IF NOT doPublish THEN
	LastPublished := 0;
	FOR i := 0 TO UsedPublishFbs - 1 DO
		PublishSendBools[i] := FALSE;
		Publishs[i](
	send:= PublishSendBools[i]);
	PublishSendFree[i] := TRUE;
	END_FOR
	
END_IF

MQTT_IN_OUT.clientFB(
	MQTT_IN_OUT:= MQTT_IN_OUT, 
	ENABLE:= TRUE, 
	URL:= broker, 
	TIMEOUT:= T#5S, 
	TLS:= FALSE);
start(CLK := working);

IF start.Q THEN
	finished := FALSE;

END_IF
IF doPublish THEN

	FOR i := 0 TO UsedPublishFbs - 1 DO
		
		IF PublishSendFree[i] AND NOT finished THEN
			PublishSendFree[i] := FALSE;
			
			//get next element
			IF LastPublished >= CountArray THEN
				finished := TRUE;
	
			ELSE
				IF TopicFix THEN
					PublishTopicStore[i] := Topic;
				ELSE
					PublishTopicStore[i] := Topic[LastPublished];	
				END_IF
				
				IF PayloadFix THEN
					PublishPayloadStore[i] := Payload;
				ELSE
					PublishPayloadStore[i] := Payload[LastPublished];	
				END_IF
				
				PublishSendBools[i] := TRUE;
			END_IF
			LastPublished := LastPublished + 1;
			
		END_IF	
		
			Publishs[i](
		Topic:=PublishTopicStore[i], 
		PayloadString:= PublishPayloadStore[i], 
		PublishAsString:= TRUE, 
		QoSIn:= QoS, 
		MRetain:= RetainIn, 
		send:= PublishSendBools[i]);
		IF Publishs[i].done THEN 
			PublishSendFree[i] := TRUE;
		END_IF
		IF Publishs[i].sendActive THEN
			PublishSendBools[i] := FALSE;
		END_IF
	END_FOR
	
END_IF

END_FUNCTION_BLOCK

// MQTT/Function/InitMQTTValue
FUNCTION InitMQTTValue : bool
VAR_INPUT
DataArray:POINTER TO CommonTypesAndFunctions.PWConfigs;
CountOfArray:UINT;
ValueToMQTTArray:POINTER TO MQTTValue;
MQTT_IN_OUT: POINTER TO MQTT_IN_OUT;
END_VAR
VAR
	i:UINT;
END_VAR

FOR i := 0 TO CountOfArray - 1 DO
	IF DataArray[i].NeedsMQTT THEN
		ValueToMQTTArray[i].Init(
			Topic:= DataArray[i].MQTTTopic, 
			ValueName:= DataArray[i].MQTTName, 
			ValuePointer:= DataArray[i].PointerTo, 
			ValueType:= DataArray[i].ValueType, 
			ValueDiff:= DataArray[i].MQTTDiff, 
			DecimalPlace:= DataArray[i].MQTTDezimal, 
			QoS:= DataArray[i].MQTTQoS, 
			RetainMqtt:= DataArray[i].MQTTRetain, 
			MinTime:= DataArray[i].MQTTTime,
			MQTT_IN_OUT:= MQTT_IN_OUT);
	END_IF
END_FOR

END_FUNCTION

// MQTT/Function Blocks/MQTTPushover
FUNCTION_BLOCK MQTTPushover
VAR_INPUT
	Data:POINTER TO PUSHOVER_DATA;
	MQTT_IN_OUT:REFERENCE TO MQTT_IN_OUT;
	CountData:UINT;
	MQTTTopic:POINTER TO STRING;
END_VAR
VAR_OUTPUT
END_VAR
VAR
	i:UINT;
	HaveToPush:BOOL;
	 
	Publish:MqttPublish;
	init:BOOL;
	PushedElement:UINT;
	SendFree: BOOL;
	// at least one message to push
	hit: BOOL;
	hitIndex:UINT;
	(*build like 'Topic(n(x)):x, Payload(n(x):x, Prio:x, Sound:x'  *)
	SendString:STRING(500);
	tmpString:STRING;
END_VAR

IF NOT init THEN
	
	init := TRUE;
	Publish.SetMqttInOut(MQTT_IN_OUT:= MQTT_IN_OUT);
END_IF
hit := FALSE;
HaveToPush := FALSE;
FOR i := 0 TO CountData - 1 DO
	IF Data[i].IsConfig THEN
		Data[i].R_T(CLK:=Data[i].Trigger^ XOR Data[i].Negate);
		IF Data[i].R_T.Q THEN
			Data[i].NeedToPush := TRUE;
		END_IF
		IF Data[i].NeedToPush THEN
			HaveToPush := TRUE;
		END_IF
		IF HaveToPush and NOT hit THEN
			hit := TRUE;
			hitIndex := i;
		END_IF
	END_IF
END_FOR

IF Publish.done THEN
	SendFree := TRUE;
END_IF


IF HaveToPush AND SendFree THEN
	SendFree := FALSE;
	//now build message
	SendString := 'Topic(';
	//add topic length
	tmpString := TO_STRING(len(Data[hitIndex].Topic^));
 	CommonTypesAndFunctions.concat(s1:= ADR(SendString), S2:=ADR(tmpString));
	//add '):'
	CommonTypesAndFunctions.concat(s1:= ADR(SendString), S2:=ADR('):'));
	//add topic
	CommonTypesAndFunctions.concat(s1:= ADR(SendString), S2:=Data[hitIndex].Topic);
	//add fixtext
	CommonTypesAndFunctions.concat(s1:= ADR(SendString), S2:=ADR(', Payload('));
	//add payload length
	tmpString := TO_STRING(len(Data[hitIndex].Payload^));
 	CommonTypesAndFunctions.concat(s1:= ADR(SendString), S2:=ADR(tmpString));
	//add '):'
	CommonTypesAndFunctions.concat(s1:= ADR(SendString), S2:=ADR('):'));
	//add topic
	CommonTypesAndFunctions.concat(s1:= ADR(SendString), S2:=Data[hitIndex].Payload);
	//add fixtext
	CommonTypesAndFunctions.concat(s1:= ADR(SendString), S2:=ADR(', Prio:'));
	//add prio
	tmpString := TO_STRING(Data[hitIndex].Prio);
 	CommonTypesAndFunctions.concat(s1:= ADR(SendString), S2:=ADR(tmpString));
	//add fixtext
	CommonTypesAndFunctions.concat(s1:= ADR(SendString), S2:=ADR(', Sound:'));
	//add prio
	tmpString := TO_STRING(Data[hitIndex].Sound);
 	CommonTypesAndFunctions.concat(s1:= ADR(SendString), S2:=ADR(tmpString));
	//done
	Data[hitIndex].NeedToPush := FALSE;
	//now send
	
END_IF

Publish(
	Topic:= MQTTTopic, 
	PayloadString:= adr(SendString), 
	PublishAsString:= TRUE, 
	QoSIn:= QoS.ExactlyOnce, 
	MRetain:= true, 
	send:= NOT SendFree);

END_FUNCTION_BLOCK

// MQTT/Function Blocks/CallbackFBs/SingelCallbacks/SingelStringCallback
FUNCTION_BLOCK SingelStringCallback IMPLEMENTS MQTT_SUBSCRIBE_CALLBACK
VAR_INPUT
END_VAR
VAR_OUTPUT
	//data was received, you have to reset this bit after checking!
	received: BOOL;
END_VAR
VAR
	MyPayload : POINTER TO STRING;
	MyTopic : POINTER TO STRING;
END_VAR

METHOD PublishReceived : BOOL
VAR_INPUT
	//Collection of received Data
	Data:CALLBACK_DATA;

END_VAR
MEM.MemMove(pSource:= Data.PayloadString, pDestination:= MyPayload, uiNumberOfBytes:= TO_UINT(data.PayloadSize + 1));
MEM.MemMove(pSource:= Data.TopicOut, pDestination:= MyTopic, uiNumberOfBytes:= CommonTypesAndFunctions.len(Data.TopicOut) + 1);

received := TRUE;
END_METHOD

METHOD Init : BOOL
VAR_INPUT
	payload:POINTER TO STRING;
	topic:POINTER TO STRING;
END_VAR
MyTopic := topic;
MyPayload := payload;
END_METHOD

METHOD ResetReceived : BOOL
VAR_INPUT
END_VAR
received := FALSE;
END_METHOD

END_FUNCTION_BLOCK

// MQTT/Function Blocks/CallbackFBs/SingelCallbacks/AllValuesCallback
(*
this FB expects all values as a string, binary receive is not suported...
Payload content is only value, no description, no special characters...
*)
FUNCTION_BLOCK AllValuesCallback IMPLEMENTS MQTT_SUBSCRIBE_CALLBACK
VAR_INPUT
END_VAR
VAR_OUTPUT
	//data was received, you have to reset this bit after checking!
	received: BOOL;

END_VAR
VAR
	VarType:IBaseLibrary.TypeClass;
	MyTarget:CommonTypesAndFunctions.ALL_TYPES_UNION_POINTER;
END_VAR

METHOD PublishReceived : BOOL
VAR_INPUT
	//Collection of received Data
	Data:CALLBACK_DATA;

END_VAR
CommonTypesAndFunctions.GetValueFromStringPt(TypeOfValue:= VarType,Target:= MyTarget, str:= DATA.PayloadString);

received := TRUE;
END_METHOD

METHOD Init : BOOL
VAR_INPUT
	SetType:IBaseLibrary.TypeClass;
	Target:CommonTypesAndFunctions.ALL_TYPES_UNION_POINTER;
END_VAR
VarType := SetType;
MyTarget := Target;
END_METHOD

METHOD ResetReceived : BOOL
VAR_INPUT
END_VAR
received := FALSE;
END_METHOD

END_FUNCTION_BLOCK

// MQTT/Function Blocks/CallbackFBs/ListCallbacks/ListAllValuesCallback
(*
this FB expects all values as a string, binary receive is not suported...
Payload content is only value, no description, no special characters...
*)
FUNCTION_BLOCK ListAllValuesCallback IMPLEMENTS MQTT_SUBSCRIBE_CALLBACK
VAR_INPUT
END_VAR
VAR_OUTPUT
END_VAR
VAR
	MyListData:POINTER TO LIST_ALLVALUES_CALLBACK_DATA;
	MyLengthOfData:ULINT;
	ListSplitTopic:BOOL;
	ListSplitPayload:BOOL;
	SplitCharPayload:BYTE;
END_VAR

METHOD PublishReceived : BOOL
VAR_INPUT
	//Collection of received Data
	Data:CALLBACK_DATA;
END_VAR

VAR
	i:ULINT;
	StrPt:POINTER TO STRING;
END_VAR
IF ListSplitTopic THEN
	//now search the right topic 
	FOR i := 0 TO MyLengthOfData - 1 DO
		IF CommonTypesAndFunctions.StrEquals(str1:= Data.TopicOutSplit^.Topics[Data.TopicOutSplit^.ValidFields - 1], str2:= MyListData[i].SubTopic) THEN
			CommonTypesAndFunctions.GetValueFromStringPt(TypeOfValue:= MyListData[i].VarTYPE ,Target:= MyListData[i].Target, str:= DATA.PayloadString);
		END_IF
	END_FOR
END_IF
IF ListSplitPayload THEN
	FOR i := 0 TO MyLengthOfData - 1 DO
		IF CommonTypesAndFunctions.StrEqualsAtStartWithDelimiter(str1:= MyListData[i].SubTopic, str2:= Data.PayloadString, delimiter:= SplitCharPayload) THEN
			//now search split char
			StrPt := Data.PayloadString;
			StrPt := StrPt + TO_DWORD(CommonTypesAndFunctions.find(str1 := StrPt, str2:= ADR(SplitCharPayload))) + 1;
			
			CommonTypesAndFunctions.GetValueFromStringPt(TypeOfValue:= MyListData[i].VarTYPE ,Target:= MyListData[i].Target, str:= StrPt);
		END_IF
	END_FOR
	
END_IF
END_METHOD

METHOD InitAsSplitTopic : BOOL
VAR_INPUT
	Data:POINTER TO LIST_ALLVALUES_CALLBACK_DATA;
	//Count of List Data
	LengthOfData:ULINT;
END_VAR
MyListData := Data;
MyLengthOfData := LengthOfData;
ListSplitTopic := TRUE;
ListSplitPayload := FALSE;
END_METHOD

(*inits FB, callback methoth then checks if the payload ist the same in the first characters as in the template
make sure to receive a string payload!
*)
METHOD InitAsSplitPayload : BOOL
VAR_INPUT
	Data:POINTER TO LIST_ALLVALUES_CALLBACK_DATA;
	//Count of List Data
	LengthOfData:ULINT;
	//spliting character
	SplitChar:BYTE;
END_VAR
MyListData :=Data;
MyLengthOfData := LengthOfData;
ListSplitTopic := FALSE;
ListSplitPayload := TRUE;
SplitCharPayload := SplitChar;
END_METHOD

END_FUNCTION_BLOCK

// MQTT/TestCases/testHighReceiveSplitPayload
FUNCTION_BLOCK testHighReceiveSplitPayload
VAR_INPUT
	Count:UINT:=TEST_TOPICS;
	broker:STRING:='test.mosquitto.org:1883';
	addTopic:STRING(200);
	repeatTime:TIME:=T#1M;
END_VAR
VAR_OUTPUT
END_VAR
VAR
	//MQTT_RECEIVE:MqttClient;
	
	
	subs:MQTTSubscribe;
	MQTT_IN_OUT_RECEIVE:MQTT_IN_OUT;
	tNewRun:TON;
	init: BOOL;
	i:UINT;
	//testTopics:ARRAY[0..TOPICS_MAX] OF STRING(255);
	testTopic:STRING:='SD_MQTT/TEST_PAYLOAD/PAYLOAD';
	testPayloadString:ARRAY[0..TOPICS_MAX]OF STRING(255);
	splitChar:STRING := '=';
	PayloadPrefix:STRING := 'Output';
	comparePayload:ARRAY[0..TOPICS_MAX]OF STRING(255);
	
	SendPayloadStorePointerArray:ARRAY[0..TOPICS_MAX] OF POINTER TO STRING;
	ReceivePayloadStore:ARRAY[0..TOPICS_MAX] OF LINT;
	SendPayloadStore:ARRAY[0..TOPICS_MAX] OF LINT;
	
	tmpString:STRING;
	tmpString2:STRING;
	step:UINT;
	subscribe: BOOL;

	HighSendPublish:HighLoadPublish;
	
	runPublishWorker: BOOL;

	
	noData: BOOL;
	nextRun: BOOL;
	ListCallback:ListAllValuesCallback;
	CallbackData:ARRAY[0..TOPICS_MAX] OF LIST_ALLVALUES_CALLBACK_DATA;
END_VAR
VAR CONSTANT
	TEST_TOPICS:UINT:= 200;
	TOPICS_MAX:UINT:=10000;
END_VAR

IF NOT init THEN
	init := TRUE;
	MQTT_IN_OUT_RECEIVE.ClientID := 'Test Client Receive';
	subs.SetMqttInOut(MQTT_IN_OUT:= MQTT_IN_OUT_RECEIVE); 
	//Testtopic();
	FOR i := 0 TO Count - 1 DO

		tmpString := PayloadPrefix;
		tmpString2 := UINT_TO_STRING(i);
		CommonTypesAndFunctions.concat(s1:= ADR(tmpString), s2:= ADR(tmpString2));
		//finished building compare payload
		comparePayload[i] := tmpString;
		CommonTypesAndFunctions.concat(s1:= ADR(tmpString), s2:= ADR(splitChar));
		SendPayloadStore[i] := i + 22;
		tmpString2 := TO_STRING(SendPayloadStore[i]);
		CommonTypesAndFunctions.concat(s1:= ADR(tmpString), s2:= ADR(tmpString2));
		//CommonTypesAndFunctions.concat(s1:= ADR(tmpString), s2:= ADR(splitChar));
		
		testPayloadString[i] := tmpString; 
		
		//compareTopic[i] := tmpString;
		CallbackData[i].SubTopic := ADR(comparePayload[i]);
		CallbackData[i].Target.POINTER_TO_LINT_T := ADR(ReceivePayloadStore[i]);
		CallbackData[i].VarTYPE := IBaseLibrary.TypeClass.TYPE_LINT;
		SendPayloadStorePointerArray[i] := ADR(testPayloadString[i]);
	END_FOR
	ListCallback.InitAsSplitPayload(Data:= ADR(CallbackData[0]), LengthOfData:= i, SplitChar:= CommonTypesAndFunctions.GetChar(splitChar));
END_IF
IF Count >= TOPICS_MAX THEN
	Count := TOPICS_MAX;
END_IF

subs(
	Subscribe:= subscribe, 
	Topic:= ADR(testTopic), 
	QoSSubscribe:= QoS.ExactlyOnce, 
	ExpectingString:= TRUE,
	Callback := ListCallback);
	
MQTT_IN_OUT_RECEIVE.clientFB(
	MQTT_IN_OUT:= MQTT_IN_OUT_RECEIVE, 
	ENABLE:= TRUE, 
	URL:= broker, 
	TIMEOUT:= T#5S, 
	TLS:= FALSE);
IF NOT MQTT_IN_OUT_RECEIVE.BROKER_CONNECTED THEN
	step := 0;
END_IF
	
HighSendPublish(
	ClientID:= 'HighSendClient', 
	Topic:= ADR(testTopic), 
	TopicFix:= TRUE, 
	payload:= ADR(SendPayloadStorePointerArray), 
	CountArray:= Count, 
	UsedPublishFbs:= 49, 
	working:= runPublishWorker, 
	broker:= broker, 
	QoS:= QoS.ExactlyOnce, 
	RetainIn:= FALSE);


CASE step OF
	0: 	step := 1;
		FOR i := 0 TO Count - 1 DO
			ReceivePayloadStore[i] := 0;
		END_FOR
	1: IF MQTT_IN_OUT_RECEIVE.BROKER_CONNECTED THEN
			step:= 5;
			//subscribe
			subscribe := TRUE;
		END_IF
	5: //wait for subscribe
		IF subs.SubscribeDone THEN
			step:= 10;
		END_IF
		 
	10: //publish all and receive data
		//start publish
		runPublishWorker := TRUE;
		step := 20;
	20: IF HighSendPublish.finished THEN
		//wait until send is done		
			runPublishWorker := FALSE;
			step:= 30;

		END_IF
	30: //now check payload
		
			noData := FALSE;
		FOR i := 0 TO Count - 1 DO
			IF ReceivePayloadStore[i] <> SendPayloadStore[i] THEN
				noData := TRUE;
				EXIT;
			END_IF
		END_FOR
		IF NOT noData THEN
			step := 40;
			//unsubscripe
			subscribe := FALSE; 
		END_IF	
	40: 
		IF nextRun OR tNewRun.Q THEN 
			nextRun := FALSE;
			step := 0;
		END_IF
END_CASE

tNewRun(in := step = 40,PT:= repeatTime);

END_FUNCTION_BLOCK

// MQTT/TestCases/testHighLoadPublish
FUNCTION_BLOCK testHighLoadPublish
VAR_INPUT
	topics:UINT:=TEST_TOPICS;
	broker:STRING:='test.mosquitto.org:1883';
	addTopic:STRING(200);
	retpeatTime:TIME:=T#1M;
END_VAR
VAR_OUTPUT
END_VAR
VAR

	HighLoad:HighLoadPublish;

	init: BOOL;
	i:UINT;
	//testTopics:ARRAY[0..TOPICS_MAX] OF STRING(255);
	testTopic:STRING(255):='High Payload Test with very very very very very very very very very very big topic/Outs';
	
	testPayload:ARRAY[0..TOPICS_MAX]OF STRING(255);
	splitChar:STRING := '=';
	PayloadPrefix:STRING := 'Output:';
	
	
	ReceivePayloadStore:ARRAY[0..TOPICS_MAX] OF LINT;
	SendPayloadStore:ARRAY[0..TOPICS_MAX] OF STRING(255);
	SendPayloadStorePointerArray:ARRAY[0..TOPICS_MAX] OF POINTER TO STRING;
	tmpString:STRING;
	tmpString2:STRING;
	step:INT;
	nextRun: BOOL;
	tNewRun:ton;
	work:BOOL;


END_VAR
VAR CONSTANT
	TEST_TOPICS:UINT:= 200;
	TOPICS_MAX:UINT:=10000;
END_VAR

IF NOT init THEN
	 init := TRUE;
	//Testtopic();
	FOR i := 0 TO topics - 1 DO
		
		tmpString := PayloadPrefix;
		tmpString2 := UINT_TO_STRING(i);
		CommonTypesAndFunctions.concat(s1:= ADR(tmpString), s2:= ADR(tmpString2));
		
		CommonTypesAndFunctions.concat(s1:= ADR(tmpString), s2:= ADR(splitChar));
		CommonTypesAndFunctions.concat(s1:= ADR(tmpString), s2:= ADR(tmpString2));
		SendPayloadStore[i] := tmpString;
		SendPayloadStorePointerArray[i] := ADR(SendPayloadStore[i]);
		step := 10;
	END_FOR
	
END_IF

HighLoad(
	ClientID:= 'Test for HighLoadPublish', 
	Topic:= ADR(testTopic), 
	TopicFix:= TRUE, 
	payload:= ADR(SendPayloadStorePointerArray[0]),
	PayloadFix := FALSE, 
	CountArray:= topics, 
	UsedPublishFbs:= MyConstants.IN_OUT_SLOTS_SIZE - 1, 
	working:= work, 
	broker:= 'windows-10-pro:1883', 
	QoS:= QoS.ExactlyOnce, 
	RetainIn:= FALSE);

IF topics >= TOPICS_MAX THEN
	topics := TOPICS_MAX - 1;
END_IF


	
CASE step OF
	10: //empty
		step := 20;
	
	20: 
		work := TRUE; 
		step := 30;
	30: //wait for finish
		IF HighLoad.finished THEN
			work := FALSE;
			step := 40;
			
		END_IF
		
	40: //wait for next run
		IF tNewRun.Q OR nextRun THEN
			step := 10;
		END_IF 
END_CASE

tNewRun(in := step = 40,PT:= retpeatTime);

END_FUNCTION_BLOCK

// MQTT/Function Blocks/CallbackFBs/Callback Collector/CallbackCollector
(*this FB collects instances of FB with the MQTT_SUBSCRIBE_CALLBACK interface.
then you can pass a instance of this FB to a subscription FB to call all of your FBs to a specific subscription topic,
in this call you can check if the packet was for your instance. If your instance methode call return true, the the FB exits the
loop an so you may save cycle time.
MEmory for instance references are created dynamic, so no restriction by library*)
FUNCTION_BLOCK CallbackCollector IMPLEMENTS MQTT_SUBSCRIBE_CALLBACK
VAR_INPUT
END_VAR
VAR_OUTPUT
END_VAR
VAR
	first:POINTER TO CALLBACK_INSTANCES := 0;
	items:UDINT;
	size:UDINT;
END_VAR

//true if all ok, else false
METHOD put : BOOL
VAR_INPUT
	instance:MQTT_SUBSCRIBE_CALLBACK;
END_VAR
VAR
	aktElement:POINTER TO CALLBACK_INSTANCES;
END_VAR
aktElement := first;

IF aktElement = 0 THEN
	//first hit...
	{info 'semaphore'}
	first := __NEW(CALLBACK_INSTANCES);
	IF first = 0 THEN
		put := FALSE;
		RETURN;
	END_IF
	aktElement := first;
ELSE
	//search last
	WHILE aktElement^.next  <> 0 DO 
		aktElement := aktElement^.next; 
	END_WHILE
	{info 'semaphore'}
	aktElement^.next := __NEW(CALLBACK_INSTANCES);
	IF aktElement^.next = 0 THEN
		put := FALSE;
		RETURN;
	END_IF
	aktElement := aktElement^.next;
END_IF

aktElement^.callback := instance;
put := TRUE;
items := items + 1;
size := size + SIZEOF(CALLBACK_INSTANCES);
END_METHOD


METHOD PublishReceived : BOOL
VAR_INPUT
	(*Collection of received Data*)
	Data	: CALLBACK_DATA;
END_VAR
VAR
	element:POINTER TO CALLBACK_INSTANCES;
	loop: BOOL := true;

END_VAR


IF first = 0 THEN
	//no callback avalable
	RETURN;
END_IF
element := first;


WHILE loop DO
	IF element^.callback.PublishReceived(Data := Data) THEN
		PublishReceived := TRUE;
		RETURN;
	END_IF
	IF element^.next = 0 THEN
		loop := FALSE;
	ELSE
		element := element^.next;
	END_IF
END_WHILE
END_METHOD

//destroy all dynamic content
METHOD destroy : BOOL
VAR_INPUT
END_VAR
VAR
	aktElement:POINTER TO CALLBACK_INSTANCES;
	nextElement:POINTER TO CALLBACK_INSTANCES;
	


END_VAR
GVL_MQTT.ProgNum := PROG_NUM.DESTROY_CALLBACK_COLLECTOR;
IF first = 0 THEN
	RETURN;
END_IF

aktElement := first;

REPEAT
	nextElement := aktElement^.next;
	__DELETE(aktElement);
	aktElement := nextElement;
	items := items - 1;
	size := size - SIZEOF(CALLBACK_INSTANCES);
UNTIL aktElement = 0
END_REPEAT
first := 0;
GVL_MQTT.ProgNum := PROG_NUM.DESTROY_CALLBACK_COLLECTOR_DONE;
END_METHOD

METHOD FB_Exit : BOOL 
VAR_INPUT 
 bInCopyCode : BOOL; // TRUE: the exit method is called in order to leave the instance which will be copied afterwards (online change). 
END_VAR
destroy();
END_METHOD

END_FUNCTION_BLOCK

// MQTT/TestCases/Test Interfaces/FooBarReceivingFB
{attribute 'reflection'}
FUNCTION_BLOCK FooBarReceivingFB IMPLEMENTS MQTT_SUBSCRIBE_CALLBACK
VAR_INPUT
END_VAR
VAR_OUTPUT
END_VAR
VAR
	{attribute 'instance-path'}
	{attribute 'noinit'}
	instanceName: STRING(255);//this string contains the instance name of the FB
	//here we get the "lowest" element of the name...
	LastTreeName:STRING;
	//if set to true we search the instance name in the lowest topic
	splitTopic: BOOL;
	//if set to true we search the instance name in Payload separatet by the split char 
	splitPayload: BOOL;
	//an this is the split char...
	SplitPayloadChar: BYTE;
	(*here is the target where we will place the payload contend
	this can be anything...*)
	Target:STRING(255);
END_VAR

METHOD PublishReceived : BOOL
VAR_INPUT
	(*Collection of received Data*)
	Data	: CALLBACK_DATA;
	
END_VAR
VAR
	StrPt : POINTER TO STRING(255);
END_VAR
// no we can check if the topic/payload fits to my instance name.... 

//now search the right topic 
IF splitTopic THEN
	
	IF CommonTypesAndFunctions.StrEquals(str1:= Data.TopicOutSplit^.Topics[Data.TopicOutSplit^.ValidFields - 1], str2:= ADR(LastTreeName)) THEN
		Target := Data.PayloadString^;
	END_IF

END_IF

//now look into the payload
IF splitPayload THEN
	
	IF CommonTypesAndFunctions.StrEqualsAtStartWithDelimiter(str1:= ADR(LastTreeName), str2:= Data.PayloadString, delimiter:= SplitPayloadChar) THEN
		//now search split char
		StrPt := Data.PayloadString;
		StrPt := StrPt + TO_DWORD(CommonTypesAndFunctions.find(str1 := StrPt, str2:= ADR(SplitPayloadChar))) + 1;
		Target := StrPt^;
	END_IF
END_IF
END_METHOD

METHOD initAsFindTopic : BOOL
VAR_INPUT
END_VAR
getLastTreeName();
splitPayload := FALSE;
splitTopic := TRUE;
END_METHOD

METHOD getLastTreeName : BOOL
VAR_INPUT
END_VAR
LastTreeName := CommonTypesAndFunctions.FindLastDot(ADR(instanceName))^;
END_METHOD

METHOD initAsFindPayload : BOOL
VAR_INPUT
	//only first char is selected
	splitChar:STRING;
END_VAR
getLastTreeName();
splitPayload := TRUE;
splitTopic := FALSE;

SplitPayloadChar := CommonTypesAndFunctions.GetChar(in:= splitChar);
END_METHOD

END_FUNCTION_BLOCK

// MQTT/TestCases/Test Interfaces/exampleForFbs
FUNCTION_BLOCK exampleForFbs
VAR_INPUT
END_VAR
VAR_OUTPUT
END_VAR
VAR
	//the MQTT client
	//client:ClientWrapper;
	//some reciving FBs
	FirstExtReceiver:FooBarReceivingFB;
	SecondExtReceiver:FooBarReceivingFB;
	ThirdExtReceiver:FooBarReceivingFB;
	FourthExtReceiver:FooBarReceivingFB;
	//a Array of receiving FBs
	ArrayReceive:ARRAY[0..9] OF FooBarReceivingFB;
	
	//the collector of the FBs
	stock:CallbackCollector;
END_VAR



(*
client(
	broker:= 'test.mosquitto.org:1883', 
	connect:= TRUE, 
	tls:= FALSE);

	*)

END_FUNCTION_BLOCK

// MQTT/Function Blocks/CallbackFBs/Callback Collector/ReceiveValueWithStrucur
FUNCTION_BLOCK ReceiveValueWithStrucur EXTENDS ReceiveValue
VAR_INPUT
END_VAR
VAR_OUTPUT
END_VAR
VAR
	InstanceName:CommonTypesAndFunctions.GetInstanceName;
	localCompString:STRING(255);
END_VAR

METHOD InitReceiveStructur : BOOL
VAR_INPUT
	
	TopicLevel:USINT;
	//this typ is my received string
	ValueTyp:CommonTypesAndFunctions.VAR_TYPES; 
	//if set to true and hit we will return true, else false...
	returnHit: BOOL;
END_VAR
VAR
	tString:STRING(255);
	cmpByte:BYTE;
	bytePointer:POINTER TO BYTE;
	StringPointer:POINTER TO STRING;
	i:UINT;
END_VAR

tString:= InstanceName.GetInstanceTopic();

cmpByte:= CommonTypesAndFunctions.GetChar('/');

bytePointer := ADR(tString) + CommonTypesAndFunctions.len(ADR(tString));

i := 0;

WHILE bytePointer >= ADR(tString) DO
	IF bytePointer^ = cmpByte THEN
		i := i + 1; 
	END_IF
	
	IF i = TopicLevel THEN
		
		StringPointer := bytePointer + 1;
		//ReceiveTopic := GVL_ZIGBEE.TextZigbeeTopic;
		//ReceiveTopic := CONCAT(STR1:= ReceiveTopic, STR2:= StringPointer^); 
		localCompString := StringPointer^;
		initAsFindTopic(compString:= ADR(localCompString), ValueTyp:= ValueTyp, returnHit:= returnHit);
		RETURN;
	END_IF
	bytePointer := bytePointer - 1;
END_WHILE
localCompString := tString;
initAsFindTopic(compString:= ADR(localCompString), ValueTyp:= ValueTyp, returnHit:= returnHit);
END_METHOD

END_FUNCTION_BLOCK

// MQTT/Function Blocks/CallbackFBs/Callback Collector/ReceiveValue
(*
Receives one value from a MQTT publish packet.
It can check diffrent sources to determinate if the data is for this Value....

*)
FUNCTION_BLOCK ReceiveValue IMPLEMENTS MQTT_SUBSCRIBE_CALLBACK
VAR_INPUT
END_VAR
VAR_OUTPUT
	//your desired payload...
	MQTTReceived:CommonTypesAndFunctions.ALL_TYPES_UNION;
	//Var was updated
	Updated: BOOL;

END_VAR
VAR
	//pointer to target
	TargetPointer:CommonTypesAndFunctions.ALL_TYPES_UNION_POINTER;
	//Target var type
	MyValueTyp:IBaseLibrary.TypeClass;
	//an this is the split char...
	SplitPayloadChar: BYTE;
	//compare with this...
	MyCompString:POINTER TO STRING;
	//and this for Payload
	MyCompStringPayload:POINTER TO STRING;
	//if set to true and hit we will return true, else false...
	MyReturnHit: BOOL;
	ReceiveType : RECEIVE_TYPS;
END_VAR


METHOD PublishReceived : BOOL
VAR_INPUT
	(*Collection of received Data*)
	Data	: CALLBACK_DATA;
END_VAR
VAR
	StrPt : POINTER TO STRING;
END_VAR
CASE ReceiveType OF
	RECEIVE_TYPS.FIND_LAST_TOPIC:	
		//now search the right topic 
		IF CommonTypesAndFunctions.StrEquals(str1:= Data.TopicOutSplit^.Topics[Data.TopicOutSplit^.ValidFields - 1], str2:= MyCompString) THEN
			CommonTypesAndFunctions.GetValueFromStringPt(TypeOfValue:= MyValueTyp ,Target:= TargetPointer, str:= DATA.PayloadString);
			PublishReceived := MyReturnHit;
			Updated := TRUE;
		END_IF
	RECEIVE_TYPS.FIND_PAYLOAD:
		IF CommonTypesAndFunctions.StrEqualsAtStartWithDelimiter(str1:= MyCompString, str2:= Data.PayloadString, delimiter:= SplitPayloadChar) THEN
			//now search split char
			StrPt := Data.PayloadString;
			StrPt := StrPt + TO_DWORD(CommonTypesAndFunctions.find(str1 := StrPt, str2:= ADR(SplitPayloadChar))) + 1;
			CommonTypesAndFunctions.GetValueFromStringPt(TypeOfValue:= MyValueTyp ,Target:= TargetPointer, str:= StrPt);
			PublishReceived := MyReturnHit;
			Updated := TRUE;
		END_IF
	RECEIVE_TYPS.FIND_LAST_TOPIC_AND_PAYLOAD:
		//now search the right topic and payload
		IF CommonTypesAndFunctions.StrEquals(str1:= Data.TopicOut, str2:= MyCompString) THEN
			IF CommonTypesAndFunctions.StrEqualsAtStartWithDelimiter(str1:= MyCompStringPayload, str2:= Data.PayloadString, delimiter:= SplitPayloadChar) THEN
				StrPt := Data.PayloadString;
				StrPt := StrPt + TO_DWORD(CommonTypesAndFunctions.find(str1 := StrPt, str2:= ADR(SplitPayloadChar))) + 1;
				CommonTypesAndFunctions.GetValueFromStringPt(TypeOfValue:= MyValueTyp ,Target:= TargetPointer, str:= StrPt);
				PublishReceived := MyReturnHit;
				Updated := TRUE;
			END_IF
		END_IF
	RECEIVE_TYPS.FIND_TOPIC:
		//now search the right topic 
		IF CommonTypesAndFunctions.StrEquals(str1:= Data.TopicOut, str2:= MyCompString) THEN
			CommonTypesAndFunctions.GetValueFromStringPt(TypeOfValue:= MyValueTyp ,Target:= TargetPointer, str:= DATA.PayloadString);
			PublishReceived := MyReturnHit;
			Updated := TRUE;
		END_IF
END_CASE
END_METHOD

METHOD initAsFindPayload : BOOL
VAR_INPUT
	//only first char is selected
	splitChar:STRING;
	//this i'm searching
	compString : POINTER TO STRING;
	//this typ is my received string
	ValueTyp:IBaseLibrary.TypeClass; 
	//if set to true and hit we will return true, else false...
	returnHit: BOOL;
END_VAR
ReceiveType := RECEIVE_TYPS.FIND_PAYLOAD;

SplitPayloadChar := CommonTypesAndFunctions.GetChar(in:= splitChar);
MyCompString := compString;
MyValueTyp := ValueTyp;
makePointer();
MyReturnHit := returnHit;
END_METHOD

(*this will only check the lowest topic level*)
METHOD initAsFindTopic : BOOL
VAR_INPUT
	//this i'm searching
	compString : POINTER TO STRING;
	//this typ is my received string
	ValueTyp:IBaseLibrary.TypeClass; 
	//if set to true and hit we will return true, else false...
	returnHit: BOOL;
END_VAR
ReceiveType := RECEIVE_TYPS.FIND_TOPIC;
MyCompString := compString;
MyValueTyp := ValueTyp;
makePointer();
MyReturnHit := returnHit;
END_METHOD

METHOD makePointer : BOOL
VAR_INPUT
END_VAR
TargetPointer := CommonTypesAndFunctions.MakeAllTypesPointer(fromWho:= adr(MQTTReceived), myType:= MyValueTyp);
END_METHOD

(*this will check the whole topic!*)
METHOD initAsFindTopicAndPayload : BOOL
VAR_INPUT
	//only first char is selected
	splitChar:STRING;
	//this topic i'm searching
	compStringTopic : POINTER TO STRING;
	//this payload i'm searching
	compStringPayload : POINTER TO STRING;
	//this typ is my received string
	ValueTyp:IBaseLibrary.TypeClass; 
	//if set to true and hit we will return true, else false...
	returnHit: BOOL;
END_VAR
ReceiveType := RECEIVE_TYPS.FIND_LAST_TOPIC_AND_PAYLOAD;
SplitPayloadChar := CommonTypesAndFunctions.GetChar(in:= splitChar);
MyCompString := compStringTopic;
MyCompStringPayload := compStringPayload;
MyValueTyp := ValueTyp;
makePointer();
MyReturnHit := returnHit;
END_METHOD

METHOD SetOutput : BOOL
VAR_INPUT
	value:CommonTypesAndFunctions.ALL_TYPES_UNION;
END_VAR
MQTTReceived := value;
END_METHOD

METHOD initAsFindLastTopic : BOOL
VAR_INPUT
	//this i'm searching
	compString : POINTER TO STRING;
	//this typ is my received string
	ValueTyp:IBaseLibrary.TypeClass; 
	//if set to true and hit we will return true, else false...
	returnHit: BOOL;
END_VAR
ReceiveType := RECEIVE_TYPS.FIND_LAST_TOPIC;
MyCompString := compString;
MyValueTyp := ValueTyp;
makePointer();
MyReturnHit := returnHit;
END_METHOD

METHOD ResetUpdate : BOOL
VAR_INPUT
END_VAR
Updated := FALSE;
END_METHOD

END_FUNCTION_BLOCK

// MQTT/Function Blocks/CallbackFBs/Callback Collector/ReceiveString
FUNCTION_BLOCK ReceiveString IMPLEMENTS MQTT_SUBSCRIBE_CALLBACK
VAR_INPUT
END_VAR
VAR_OUTPUT
	//your desired payload...
	MQTTReceived:STRING(255);
END_VAR
VAR
	//if set to true we search the instance name in the lowest topic
	splitTopic: BOOL;
	//if set to true we search the instance name in Payload separatet by the split char 
	splitPayload: BOOL;
	//an this is the split char...
	SplitPayloadChar: BYTE;
	//compare with this...
	MyCompString:POINTER TO STRING;
	//if set to true and hit we will return true, else false...
	MyReturnHit: BOOL;
END_VAR

METHOD PublishReceived : BOOL
VAR_INPUT
	(*Collection of received Data*)
	Data	: CALLBACK_DATA;
	
END_VAR
VAR
	StrPt : POINTER TO STRING(255);
END_VAR
// no we can check if the topic/payload matches to my compare string 

//now search the right topic 
IF splitTopic THEN
	
	IF CommonTypesAndFunctions.StrEquals(str1:= Data.TopicOut, str2:= MyCompString) THEN
		StrPt := Data.PayloadString;
		MQTTReceived := StrPt^;
		PublishReceived := MyReturnHit;
	END_IF

END_IF

//now look into the payload
IF splitPayload THEN
	
	IF CommonTypesAndFunctions.StrEqualsAtStartWithDelimiter(str1:= MyCompString, str2:= Data.PayloadString, delimiter:= SplitPayloadChar) THEN
		//now search split char
		StrPt := Data.PayloadString;
		StrPt := StrPt + TO_DWORD(CommonTypesAndFunctions.find(str1 := StrPt, str2:= ADR(SplitPayloadChar))) + 1;
		MQTTReceived := StrPt^;
		PublishReceived := MyReturnHit;
	END_IF
END_IF
END_METHOD

METHOD initAsFindTopic : BOOL
VAR_INPUT
	//this i'm searching
	compString : POINTER TO STRING;
	//if set to true and hit we will return true, else false...
	returnHit: BOOL;
END_VAR

splitPayload := FALSE;
splitTopic := TRUE;
MyCompString := compString;
MyReturnHit := returnHit;
END_METHOD

METHOD initAsFindPayload : BOOL
VAR_INPUT
	//only first char is selected
	splitChar:STRING;
	//this i'm searching
	compString : POINTER TO STRING;
	//if set to true and hit we will return true, else false...
	returnHit: BOOL;
END_VAR

splitPayload := TRUE;
splitTopic := FALSE;

SplitPayloadChar := CommonTypesAndFunctions.GetChar(in:= splitChar);
MyCompString := compString;
MyReturnHit := returnHit;
END_METHOD

END_FUNCTION_BLOCK

// MQTT/TestCases/TestLongPublish
FUNCTION_BLOCK TestLongPublish
VAR_INPUT
	broker:STRING := 'test.mosquitto.org:1883';
END_VAR
VAR_OUTPUT
END_VAR
VAR
	longPayload:STRING(8000):='';
	longTopic:STRING(8000):=('TestTopic/');
	longPayloadReceive:STRING(8000);
	longTopicReceive:STRING(8000);
	init: BOOL;
	i1:UINT;
	i2:UINT;
	countAsciis :UINT := 48;
	pt1:POINTER TO BYTE;
	pt2:POINTER TO BYTE;
	
	step : UINT; 
	
	//MQTT:MqttClient;
	
	MQTT_IN_OUT:MQTT_IN_OUT;
	
	ComConfig:COM_CONFIG;
	
	pup:MqttPublish;
	send: BOOL;

	
	SUB1:MQTTSubscribe;
	subscribe: BOOL;

	callback : SingelStringCallback;
	
	
	connect: BOOL;

	nextRung:ton;
	lenPayload:UINT;
	lenTopic:uint;
	
END_VAR

IF NOT init THEN
	init := TRUE;
	SUB1.SetMqttInOut(MQTT_IN_OUT := MQTT_IN_OUT);
	pup.SetMqttInOut(MQTT_IN_OUT := MQTT_IN_OUT);
	ComConfig.MaxPayloadSize := 20000;
	ComConfig.MaxTopicLevels := 10;
	ComConfig.MaxTopicElementSize := 10000;
	
	MQTT_IN_OUT.ClientID := 'TestCodesys';
	MQTT_IN_OUT.COM_CONFIG := ComConfig;
	//firs build some nice pacload ...
	pt1 := ADR(longPayload);
	pt2 := ADR(longTopic);
	pt2 := pt2 + 10;
	FOR i1 := 0 TO 8000 / countAsciis - 1 DO
		FOR i2 := 0 TO countAsciis - 1 DO
			pt1^ := TO_BYTE(i2 + 16#30); //16#30 --> ASCII zero
			pt2^ := TO_BYTE(i2 + 16#30); //16#30 --> ASCII zero
			pt1 := pt1 + 1;
			pt2 := pt2 + 1;
		END_FOR
	END_FOR
	//need termination...
	pt1^:= 0;
	pt2^:= 0;
	callback.Init(payload:= ADR(longPayloadReceive), topic:= ADR(longTopicReceive));
END_IF

SUB1(
	Subscribe:= subscribe, 
	Topic:= ADR('TestTopic/#'), 
	QoSSubscribe:= QoS.ExactlyOnce, 
	ExpectingString:= TRUE, 
	Callback:= callback);

	
	pup(
	Topic:= ADR(longTopic), 
	PayloadString:= ADR(longPayload), 
	PublishAsString:= TRUE, 
	QoSIn:= Qos.ExactlyOnce, 
	MRetain:= FALSE, 
	send:= send);

MQTT_IN_OUT.clientFB(
	MQTT_IN_OUT:= MQTT_IN_OUT, 
	ENABLE:= connect, 
	URL:= broker, 
	TIMEOUT:= T#5S);


CASE step OF 
	0://begin
		//connect
		connect := TRUE;
		step := 10;
	10://wait connected
		IF MQTT_IN_OUT.BROKER_CONNECTED THEN
			//subscribe
			subscribe := TRUE;		
			step := 20;
		END_IF
	20://wait subscribed
		IF SUB1.SubscribeDone THEN
			//send packet and check receive
			send := TRUE;
			step := 30;
		END_IF
		
	30:
		//reset send
		send := FALSE;
		step := 40;
	40:
		lenPayload:= CommonTypesAndFunctions.len(ADR(longPayloadReceive));
		lenTopic:= CommonTypesAndFunctions.len(ADR(longTopicReceive));
		//check if payload and topic received....
		IF CommonTypesAndFunctions.StrEquals(str1:= ADR(longPayload), str2:= ADR(longPayloadReceive)) AND
			CommonTypesAndFunctions.StrEquals(str1:= ADR(longTopic), str2:= ADR(longTopicReceive)) THEN
			//deled received strings
			longTopicReceive := '';
			longPayloadReceive := '';
			//go wait repeat
			step := 50;
		END_IF
		
	50:
		IF nextRung.Q THEN
			step := 0;
		END_IF
END_CASE

nextRung(IN:= step = 50, PT:= T#5S);

END_FUNCTION_BLOCK

// MQTT/TestCases/TestLongStringList
FUNCTION_BLOCK TestLongStringList
VAR_INPUT
	//use this input if you want to test with another broker
	client:STRING:='test.mosquitto.org:1883';//test.mosquitto.org
	
END_VAR
VAR_OUTPUT
END_VAR
VAR
	//MQTTClient:MqttClient;
	MQTT_IN_OUT:MQTT_IN_OUT;
	MQTTInfo:MQTT_INFO;
	publish:MqttPublish;
	subscribe:MQTTSubscribe;
	ReceiveSubscribeTopic:STRING(255);
	
	ReceiveSubscribePayloadLong:STRING(500);
	State :MQTTState;
	init: BOOL;
	varSend: BOOL;
	timerSend:ton;
	t1:ton;
	t2:ton;
	Payload:STRING;
	//the method PublishReceved() is call when an publsih packet form the broker is received.
	StringCallback:ListStringCallback;
	//the array contains the targets and sub topics for receive
	CallBackTargets:ARRAY[0..1] OF LIST_STRING_CALLBACK_DATA := [(Target:=ADR(ReceiveSubscribePayloadLong), SubTopic:= ADR('Long'))];
	len1:UINT;
END_VAR

//here init is done
IF NOT init THEN
	init := TRUE;
	MQTT_IN_OUT.ClientID := CONCAT('CodesysMqtt',TO_STRING(TICKS.GetTick(xDummy:= TRUE)));
	//init state FB, so you only have to call state();without parameters... 
	State.Init(
	State:= ADR(t1.Q), 
	Topic:= ADR('CODESYS-MQTT-BY-SD/Long'), 
	StateName:= ADR(''), 
	StateValueOn:= ADR('LOOOOOOOOOOOOOOOOOOOOOOOOOOOOOOOOOOOOOOOOOOOOOOOOOOOOOOOOOOOOOOOOOOOOOOOOOOOOOOOOOOOOOOOOOOOOOOOOOOOOOOOOOOOOOOOOOOOOOOOOOOOOOOOOOOOOOOOOOOOOOOOOOOOOOOOOOOOOOOOOOOOOOOOOOOOOOOOOOOOOOOOOOOOOOOOOOOOOOOOOOOOOOOOOOOOOOOOOg:On'), 
	StateValueOff:= ADR('LOOOOOOOOOOOOOOOOOOOOOOOOOOOOOOOOOOOOOOOOOOOOOOOOOOOOOOOOOOOOOOOOOOOOOOOOOOOOOOOOOOOOOOOOOOOOOOOOOOOOOOOOOOOOOOOOOOOOOOOOOOOOOOOOOOOOOOOOOOOOOOOOOOOOOOOOOOOOOOOOOOOOOOOOOOOOOOOOOOOOOOOOOOOOOOOOOOOOOOOOOOOOOOOOOOOOOOOOg:Off'), 
	QoS:= QoS.ExactlyOnce, 
	RetainMqtt:= TRUE,
	MQTT_IN_OUT:= MQTT_IN_OUT);
	StringCallback.InitAsSplitTopic(ListData := ADR(CallBackTargets), LengthOfData:= 1);
	
	subscribe.SetMqttInOut(MQTT_IN_OUT:= MQTT_IN_OUT);
	
END_IF
//timer for repeating packets
t1(IN:= NOT t2.Q, PT:= T#1S, );
t2(IN:= t1.Q, PT:= T#1S);
//call of MQTT client
MQTT_IN_OUT.clientFB(
	MQTT_IN_OUT:= MQTT_IN_OUT, 
	ENABLE:= TRUE, 
	URL:= client, 
	TIMEOUT:= T#5S, 
	TLS:= FALSE);
//Subscribe to topic
subscribe(
	Subscribe:= TRUE, 
	Topic:= ADR('CODESYS-MQTT-BY-SD/#'), 
	QoSSubscribe:= QoS.ExactlyOnce, 
	ExpectingString:= TRUE,
	Callback:= StringCallback);
len1 := CommonTypesAndFunctions.len(str:= ADR(ReceiveSubscribePayloadLong));

//call of state FB
State();

END_FUNCTION_BLOCK

// MQTT/TestCases/TestStringPointer
FUNCTION_BLOCK TestStringPointer
VAR_INPUT
END_VAR
VAR_OUTPUT
END_VAR
VAR
	SFrom:STRING(2000):='ABCDEFGHIJKLMNOPQRSTUVWXYZABCDEFGHIJKLMNOPQRSTUVWXYZABCDEFGHIJKLMNOPQRSTUVWXYZABCDEFGHIJKLMNOPQRSTUVWXYZABCDEFGHIJKLMNOPQRSTUVWXYZABCDEFGHIJKLMNOPQRSTUVWXYZABCDEFGHIJKLMNOPQRSTUVWXYZABCDEFGHIJKLMNOPQRSTUVWXYZABCDEFGHIJKLMNOPQRSTUVWXYZABCDEFGHIJKLMNOPQRSTUVWXYZABCDEFGHIJKLMNOPQRSTUVWXYZABCDEFGHIJKLMNOPQRSTUVWXYZABCDEFGHIJKLMNOPQRSTUVWXYZABCDEFGHIJKLMNOPQRSTUVWXYZABCDEFGHIJKLMNOPQRSTUVWXYZABCDEFGHIJKLMNOPQRSTUVWXYZABCDEFGHIJKLMNOPQRSTUVWXYZABCDEFGHIJKLMNOPQRSTUVWXYZABCDEFGHIJKLMNOPQRSTUVWXYZABCDEFGHIJKLMNOPQRSTUVWXYZABCDEFGHIJKLMNOPQRSTUVWXYZABCDEFGHIJKLMNOPQRSTUVWXYZABCDEFGHIJKLMNOPQRSTUVWXYZABCDEFGHIJKLMNOPQRSTUVWXYZABCDEFGHIJKLMNOPQRSTUVWXYZABCDEFGHIJKLMNOPQRSTUVWXYZABCDEFGHIJKLMNOPQRSTUVWXYZABCDEFGHIJKLMNOPQRSTUVWXYZABCDEFGHIJKLMNOPQRSTUVWXYZABCDEFGHIJKLMNOPQRSTUVWXYZABCDEFGHIJKLMNOPQRSTUVWXYZABCDEFGHIJKLMNOPQRSTUVWXYZABCDEFGHIJKLMNOPQRSTUVWXYZABCDEFGHIJKLMNOPQRSTUVWXYZABCDEFGHIJKLMNOPQRSTUVWXYZABCDEFGHIJKLMNOPQRSTUVWXYZABCDEFGHIJKLMNOPQRSTUVWXYZABCDEFGHIJKLMNOPQRSTUVWXYZABCDEFGHIJKLMNOPQRSTUVWXYZABCDEFGHIJKLMNOPQRSTUVWXYZABCDEFGHIJKLMNOPQRSTUVWXYZABCDEFGHIJKLMNOPQRSTUVWXYZABCDEFGHIJKLMNOPQRSTUVWXYZABCDEFGHIJKLMNOPQRSTUVWXYZABCDEFGHIJKLMNOPQRSTUVWXYZABCDEFGHIJKLMNOPQRSTUVWXYZABCDEFGHIJKLMNOPQRSTUVWXYZABCDEFGHIJKLMNOPQRSTUVWXYZABCDEFGHIJKLMNOPQRSTUVWXYZABCDEFGHIJKLMNOPQRSTUVWXYZABCDEFGHIJKLMNOPQRSTUVWXYZABCDEFGHIJKLMNOPQRSTUVWXYZABCDEFGHIJKLMNOPQRSTUVWXYZABCDEFGHIJKLMNOPQRSTUVWXYZABCDEFGHIJKLMNOPQRSTUVWXYZABCDEFGHIJKLMNOPQRSTUVWXYZABCDEFGHIJKLMNOPQRSTUVWXYZABCDEFGHIJKLMNOPQRSTUVWXYZABCDEFGHIJKLMNOPQRSTUVWXYZABCDEFGHIJKLMNOPQRSTUVWXYZABCDEFGHIJKLMNOPQRSTUVWXYZABCDEFGHIJKLMNOPQRSTUVWXYZABCDEFGHIJKLMNOPQRSTUVWXYZABCDEFGHIJKLMNOPQRSTUVWXYZABCDEFGHIJKLMNOPQRSTUVWXYZABCDEFGHIJKLMNOPQRSTUVWXYZABCDEFGHIJKLMNOPQRSTUVWXYZABCDEFGHIJKLMNOPQRSTUVWXYZ';
	STo:STRING(1000):='';
	p1:POINTER TO STRING(2000);
	p2:POINTER TO STRING(2000);
	l1:UINT;
	l2:UINT;
END_VAR

l1 := CommonTypesAndFunctions.len(str:= ADR(SFrom));
l2 := CommonTypesAndFunctions.len(str:= ADR(STo));
p1:= ADR(SFrom);
p2:= ADR(STo);
p2^:= p1^;

END_FUNCTION_BLOCK

// MQTT/TestCases/TestUserPassword
FUNCTION_BLOCK TestUserPassword
VAR_INPUT
END_VAR
VAR_OUTPUT
END_VAR
VAR
MQTT1:MqttClient ;
MQTT2:MqttClient ;
MQTT3:MqttClient ;	
info:MQTT_INFO;
MQTT_IN_OUT:MQTT_IN_OUT;
END_VAR

MQTT1(MQTT_IN_OUT := MQTT_IN_OUT,
	ENABLE := TRUE,
	URL:= 'User1:Mypassword@test.mosquitto.org:1883');
	
MQTT2(MQTT_IN_OUT := MQTT_IN_OUT,
	ENABLE := TRUE,
	URL:= 'User1@test.mosquitto.org:1883');
	
MQTT3(MQTT_IN_OUT := MQTT_IN_OUT,
	ENABLE := TRUE,
	URL:= 'User2:Mypassword@test.mosquitto.org:1883');

END_FUNCTION_BLOCK

// MQTT/Function Blocks/CallbackFBs/Callback Collector/ReceiverBase
FUNCTION_BLOCK ReceiverBase
VAR_INPUT
END_VAR
VAR_OUTPUT
END_VAR
VAR
	MatchTyp:RECEIVER_INIT_TYPS;
	Target:CommonTypesAndFunctions.ALL_TYPES_UNION_POINTER;
	TargetType:IBaseLibrary.TypeClass;
	PayloadCompare:POINTER TO STRING;
	TopicCompare:POINTER TO STRING;
	delimiter:BYTE;
	delimiterString:STRING(3);
	SplitTopic:HandleSplitTopic;
END_VAR

METHOD init
VAR_INPUT
	MQTT_IN_OUT:POINTER TO MQTT_IN_OUT;
	MatchTyp:RECEIVER_INIT_TYPS;
	Target:CommonTypesAndFunctions.ALL_TYPES_UNION_POINTER;
	TargetType:IBaseLibrary.TypeClass;
	PayloadCompare:POINTER TO STRING;
	TopicCompare:POINTER TO STRING;
	delimiter:BYTE;
	
END_VAR
MatchTyp := MatchTyp;
Target := Target;
TargetType := TargetType;
PayloadCompare := PayloadCompare;
TopicCompare := TopicCompare;
delimiter := delimiter;
delimiterString[0] := delimiter;
delimiterString[1] := 0;

IF MatchTyp = RECEIVER_INIT_TYPS.MQTT_STRING or MatchTyp = RECEIVER_INIT_TYPS.MQTT_STRING_JSON THEN
	SplitTopic.LowInit(TopicsLevelInit:= MQTT_IN_OUT^.COM_CONFIG.MaxTopicLevels,
			 SplitElementSizeInit:= MQTT_IN_OUT^.COM_CONFIG.MaxTopicElementSize, dynMemUsageInit:= ADR(MQTT_IN_OUT^.dynMemUsage));
	SplitTopic.NewTopic(in:= TopicCompare, test:= TRUE, SizeOfString:= CommonTypesAndFunctions.len(str:= TopicCompare));
END_IF
END_METHOD

METHOD CheckMatch : BOOL
VAR_INPUT
	(*Collection of received Data*)
	Data	: CALLBACK_DATA;
END_VAR
VAR 
	foundPos:DINT;
END_VAR
CheckMatch := FALSE;
CASE MatchTyp OF
	RECEIVER_INIT_TYPS.FIND_FULL_TOPIC:
		IF CommonTypesAndFunctions.StrEquals(str1:= Data.TopicOut , str2:= PayloadCompare) THEN
			CheckMatch := TRUE;
			GetValue(fromWhere:= Data.PayloadString);
			RETURN;
		END_IF 
	RECEIVER_INIT_TYPS.FIND_LAST_TOPIC:
		IF CommonTypesAndFunctions.StrEquals(str1:= Data.TopicOutSplit^.Topics[Data.TopicOutSplit^.ValidFields - 1], str2:= PayloadCompare) THEN
			CheckMatch := TRUE;
			GetValue(fromWhere:= Data.PayloadString);
			RETURN;
		END_IF
	RECEIVER_INIT_TYPS.FIND_PAYLOAD:
		IF CommonTypesAndFunctions.StrEqualsAtStartWithDelimiter(str1:= PayloadCompare, str2:= Data.PayloadString , delimiter:= delimiter) THEN
			CheckMatch := TRUE;
			GetValue(fromWhere:= Data.PayloadString + TO_UINT(CommonTypesAndFunctions.find(str1:= Data.PayloadString, str2:= ADR(delimiterString)))+1);
			RETURN;	
		END_IF
	RECEIVER_INIT_TYPS.JSON_FULL:
		IF CommonTypesAndFunctions.StrEquals(str1:= Data.TopicOut , str2:= PayloadCompare) THEN
			foundPos := CommonTypesAndFunctions.find(str1:= Data.PayloadString, str2:= TopicCompare); 
			IF foundPos >= 0 THEN
				CheckMatch := TRUE;
				RETURN;	
			END_IF
		END_IF
	RECEIVER_INIT_TYPS.JSON_SMALL:
		IF CommonTypesAndFunctions.StrEquals(str1:= Data.TopicOutSplit^.Topics[Data.TopicOutSplit^.ValidFields - 1], str2:= PayloadCompare) THEN
			IF CommonTypesAndFunctions.find(str1:= Data.PayloadString, str2:= TopicCompare) >= 0 THEN
				CheckMatch := TRUE;
				RETURN;	
			END_IF
		END_IF
	RECEIVER_INIT_TYPS.MQTT_STRING:
		IF SplitTopic.CheckTopicMatchToMe(with:= Data.TopicOutSplit) = TOPIC_MATCH.TOPIC_MATCHES THEN
			CheckMatch := TRUE;
			RETURN;
		END_IF
	RECEIVER_INIT_TYPS.MQTT_STRING_JSON:
		IF SplitTopic.CheckTopicMatchToMe(with:= Data.TopicOutSplit) = TOPIC_MATCH.TOPIC_MATCHES THEN
			IF CommonTypesAndFunctions.find(str1:= Data.PayloadString, str2:= TopicCompare) >= 0 THEN
				CheckMatch := TRUE;
				RETURN;	
			END_IF
		END_IF
	
END_CASE
END_METHOD

METHOD GetValue
VAR_INPUT
	fromWhere: POINTER TO STRING(65000);
END_VAR
CASE TargetType OF
	IBaseLibrary.TypeClass.TYPE_BOOL,
	IBaseLibrary.TypeClass.TYPE_BYTE,
	IBaseLibrary.TypeClass.TYPE_DATE,
	IBaseLibrary.TypeClass.TYPE_DINT,
	IBaseLibrary.TypeClass.TYPE_DATEANDTIME,
	IBaseLibrary.TypeClass.TYPE_DWORD,
	IBaseLibrary.TypeClass.TYPE_INT,
	IBaseLibrary.TypeClass.TYPE_LINT,
	IBaseLibrary.TypeClass.TYPE_LREAL,
	IBaseLibrary.TypeClass.TYPE_LWORD,
	IBaseLibrary.TypeClass.TYPE_REAL,
	IBaseLibrary.TypeClass.TYPE_SINT,
	IBaseLibrary.TypeClass.TYPE_TIME,
	IBaseLibrary.TypeClass.TYPE_TIMEOFDAY ,
	IBaseLibrary.TypeClass.TYPE_UDINT,
	IBaseLibrary.TypeClass.TYPE_UINT,
	IBaseLibrary.TypeClass.TYPE_ULINT,
	IBaseLibrary.TypeClass.TYPE_USINT,
	IBaseLibrary.TypeClass.TYPE_WORD:
	CommonTypesAndFunctions.GetValueFromStringPt
				(TypeOfValue:= TargetType, Target:= Target, str:= fromWhere);
END_CASE
//This was a typ too
//IBaseLibrary.TypeClass. TYPE_TOD2,
END_METHOD

END_FUNCTION_BLOCK

// MQTT/TestCases/Test Interfaces/TestCallbackCollecktor
FUNCTION_BLOCK TestCallbackCollecktor
VAR_INPUT
END_VAR
VAR_OUTPUT
END_VAR
VAR
	var1:AllValuesCallback;
	var2:AllValuesCallback;
	var3:AllValuesCallback;
	collector:CallbackCollector;
	init: BOOL;
	target1:INT;
	pt1:CommonTypesAndFunctions.ALL_TYPES_UNION_POINTER;
	callbackData:CALLBACK_DATA;
	stringPayload:STRING :='123';
END_VAR

IF NOT init THEN
	init := TRUE;
	pt1.POINTER_TO_INT_T := ADR(target1);
	var1.Init(SetType := IBaseLibrary.TypeClass.TYPE_INT, Target := pt1);
	callbackData.PayloadString := ADR(stringPayload);
END_IF

//try delet without registert instance
collector.destroy();
//put one instance
collector.put(instance:= var1);

collector.PublishReceived(Data:= callbackData);

collector.destroy();

//put two instance
collector.put(instance:= var1);
collector.put(instance:= var1);

collector.PublishReceived(Data:= callbackData);

collector.destroy();

//put tree instance
collector.put(instance:= var1);
collector.put(instance:= var1);
collector.put(instance:= var1);

collector.PublishReceived(Data:= callbackData);

collector.destroy();

//put tree instance
collector.put(instance:= var1);
collector.put(instance:= var2);
collector.put(instance:= var3);

METHOD FB_Exit : BOOL
VAR_INPUT 
 bInCopyCode : BOOL; // TRUE: the exit method is called in order to leave the instance which will be copied afterwards (online change). 
END_VAR
collector.destroy();
END_METHOD

END_FUNCTION_BLOCK

// MQTT/TestCases/TestMemHandle
FUNCTION_BLOCK TestMemHandle
VAR_INPUT
END_VAR
VAR_OUTPUT
END_VAR
VAR
	MQTT_IN_OUT_1:MQTT_IN_OUT;
	MQTT_IN_OUT_2:MQTT_IN_OUT;
	//Client1:MqttClient;
	//Client2:MqttClient;
END_VAR

MQTT_IN_OUT_1.clientFB(
	MQTT_IN_OUT:= MQTT_IN_OUT_1, 
	ENABLE:= TRUE, 
	URL:= 'test.mosquitto.org:1883', 
	TIMEOUT:= T#5S);
	
MQTT_IN_OUT_2.clientFB(
	MQTT_IN_OUT:= MQTT_IN_OUT_2, 
	ENABLE:= TRUE, 
	URL:= 'test.mosquitto.org:1883', 
	TIMEOUT:= T#5S);

END_FUNCTION_BLOCK

// MQTT/TestCases/TestSplitTopic
FUNCTION_BLOCK TestSplitTopic
VAR_INPUT
END_VAR
VAR_OUTPUT
END_VAR
VAR
	Split1:HandleSplitTopic;
	Split2:HandleSplitTopic;
	Usage1:UDINT;
	Usage2:UDINT;
	COM_CONFIG:COM_CONFIG;
END_VAR

Split1.FullInit(TopicsLevelInit:= COM_CONFIG.MaxTopicLevels, SplitElementSizeInit:= COM_CONFIG.MaxTopicElementSize, dynMemUsageInit:= ADR(Usage1));
Split2.LowInit(TopicsLevelInit:= COM_CONFIG.MaxTopicLevels, SplitElementSizeInit:= COM_CONFIG.MaxTopicElementSize, dynMemUsageInit:= ADR(Usage1));

Split1.destroy();
Split2.destroy();

END_FUNCTION_BLOCK

// MQTT/TestCases/testLongTime
FUNCTION_BLOCK testLongTime
VAR_INPUT
	client:STRING:='broker.hivemq.com';
	enable:BOOL:=TRUE;
	MyQoS:QoS:= QoS.ExactlyOnce;
END_VAR
VAR_OUTPUT
	MQTT_IN_OUT:POINTER TO MQTT_IN_OUT;
END_VAR
VAR
	//mqtt:MqttClient;
	in_out:MQTT_IN_OUT;
	init: BOOL;
	publisher:ARRAY[0..49] OF MqttPublish;
	topics:ARRAY[0..49] OF STRING(255);
	payloads:ARRAY[0..49] OF STRING;
	receiver:ARRAY[0..49] OF ReceiveValue;
	collector:CallbackCollector;
	subscriber:MQTTSubscribe;
	i:INT;
	fbRand:CommonTypesAndFunctions.Rand;
	RTCon:R_TRIG;
	worker:INT := 45;
END_VAR

IF NOT init THEN
	init := TRUE;
	FOR i := 0 TO 49 DO
		collector.put(receiver[i]);
		publisher[i].SetMqttInOut(MQTT_IN_OUT:= in_out);
		publisher[i].send := TRUE;
		payloads[i] := TO_STRING(i);
		topics[i] := CONCAT(STR1:='TestTopic/',STR2:= CONCAT(STR1:= TO_STRING(i), STR2:='/data'));
		receiver[i].initAsFindTopic(compString:=ADR(topics[i]),returnHit := TRUE,ValueTyp:= IBaseLibrary.TypeClass.TYPE_REAL);
	END_FOR
	subscriber.SetMqttInOut(MQTT_IN_OUT:= in_out);
	in_out.ClientID := 'TestLongTimeSD';
END_IF
RTCon(CLK:= in_out.BROKER_CONNECTED);
IF RTCon.Q THEN
	FOR i:=0 TO 49 DO
		publisher[i].send := TRUE;
	END_FOR
END_IF

in_out.clientFB(
	MQTT_IN_OUT:= in_out, 
	ENABLE:= enable, 
	URL:= client, 
	TIMEOUT:= T#5S);
	
subscriber(
	Subscribe:= TRUE, 
	Topic:= ADR('TestTopic/#'), 
	QoSSubscribe:= MyQoS, 
	ExpectingString:= TRUE, 
	Callback:= collector);
	
FOR i := 0 TO worker DO
	
	IF publisher[i].done THEN
		
		payloads[i] := TO_STRING(fbRand.getRand(LowIn:=1, HighIn:=1000)/10.0);
		publisher[i].send := TRUE;
	END_IF
	publisher[i](
	Topic:= ADR(topics[i]), 
	PayloadString:= ADR(payloads[i]), 
	PublishAsString:= TRUE,
	QoSIn:= MyQoS, 
	MRetain:= FALSE);
	publisher[i].send := FALSE;
END_FOR

//FB_Init ist immer implizit verfügbar und wird primär für die Initialisierung verwendet.
//Der Rückgabewert wird nicht ausgewertet. Für gezielte Einflussnahme können Sie
//die Methoden explizit deklarieren und darin mit dem Standard-Initialisierungscode 
//zusätzlichen Code bereitstellen. Sie können den Rückgabewert auswerten.
METHOD FB_Init: BOOL
VAR_INPUT    
bInitRetains: BOOL; // TRUE: Die Retain-Variablen werden initialisiert (Reset warm / Reset kalt)    
bInCopyCode: BOOL;  // TRUE: Die Instanz wird danach in den Kopiercode kopiert (Online-Change)
END_VAR
MQTT_IN_OUT := adr(in_out);
END_METHOD

END_FUNCTION_BLOCK

// MQTT/Function Blocks/Supvervision/MQTTSupvervision
(*publishs some might usefull data to your broker,
call this after your handle if you want to use the url of your conrolled cliente-broker*)
FUNCTION_BLOCK MQTTSupvervision
VAR_INPUT
	who:MQTT_IN_OUT;
	//this the X Time, send the data after x seconds, for good resaults use whole multiplrs of your cycle time
	TimeX:TIME:=T#100MS;
	//broker, if broker is different to watched broker
	broker:STRING;
END_VAR
VAR_OUTPUT
END_VAR
VAR
	init: BOOL;
	MQTT_IN_OUT:MQTT_IN_OUT;
	//handle:MqttClient;
	aktData:SUPERVISION_DATA;
	LastData:COUNTING_DATAS;
	all:CommonTypesAndFunctions.ALL_TYPES_UNION;
	i:UINT;
	publisher:ARRAY[0..COUNT_PUBLISHER] OF MQTTValue;
	HistoryPublisher:MqttPublish;
	topics:ARRAY[0..COUNT_PUBLISHER] OF STRING;
	lBroker:STRING;
	SendedBytesPerSecond:UDINT;
	SendedBytesPerSecondLast:ULINT;
	SendedBytesPerX:UDINT;
	SendedBytesPerXLast:ULINT;
	
	ReceivedBytesPerSecond:UDINT;
	ReceivedBytesPerSecondLast:ULINT;
	ReceivedBytesPerX:UDINT;
	ReceivedBytesPerXLast:ULINT;
	PublishSendPerX:UINT;
	PublishSendPerXLast:ULINT;
	PublishReceivedPerX:UINT;
	PublishReceivedPerXLast:ULINT;
	
	OldHistoryNum:UINT;
	HistoryJSON:SUPERVISION_HISTORY;
	toJSON:PRO_JSON.STRUCT_TO_JSON;
	HistoryTopic:STRING;
	HistoryString:STRING(255);
	SendHistroy: BOOL;
	LastHistoryFound: BOOL;
	tc : TIME;
	tx: DWORD;
	tl: DWORD;
	TriggerX: BOOL;
	perXTopic:STRING(10);
END_VAR
VAR_TEMP
	TempString:STRING(200);
END_VAR
VAR CONSTANT
	COUNT_PUBLISHER:UINT:=50;
END_VAR

(* measure cycle time tc and make sure this circuitry is not called more then once in x ms*)
tx := OSCAT_BASIC.T_PLC_MS();
IF NOT init THEN
	init := TRUE;
	tl := tx;
	MQTT_IN_OUT.ClientID := concat(STR1:= who.ClientID, STR2:= 'Supervisor');
	MQTT_IN_OUT.COM_CONFIG.CountSlotsIn := 10;
	MQTT_IN_OUT.COM_CONFIG.CountSlotsOut := 50;
	MQTT_IN_OUT.COM_CONFIG.MaxTopicLevels := 5;
	MQTT_IN_OUT.COM_CONFIG.MaxTopicElementSize := 100;
	MQTT_IN_OUT.doHistory := FALSE;
	IF len(broker) = 0 THEN
		lBroker := who.clientFB.URL;
	ELSE
		lBroker := broker;
	END_IF
	HistoryPublisher.SetMqttInOut(MQTT_IN_OUT:= MQTT_IN_OUT);
	HistoryTopic := concat(STR1:= who.ClientID,STR2:='Supervision/History');
	HistoryJSON.when.AsString := 'DT';
	aktData := who.clientFB.GetSupervision();
	
	//build Topics
	perXTopic := TO_STRING(TimeX);
	//replace wildcard #
	perXTopic := OSCAT_BASIC.REPLACE_ALL(str:= perXTopic, src:='#', rep:='');
	topics[0] := concat(STR1:= who.ClientID,STR2:='Supervision/RepeatedPublish');
	publisher[0].InitAny(who:= aktData.counts^.RepeatedPublish,	Topic:= ADR(topics[0]), ValueName:= ADR(''), ValueDiff:= 0, DecimalPlace:= 0, QoS:= QoS.AtMostOnce, RetainMqtt:= TRUE, MinTime:= T#1S, MQTT_IN_OUT:= MQTT_IN_OUT);
	topics[1] := concat(STR1:= who.ClientID,STR2:='Supervision/RepeatedPublishsAfterPubrel');
	publisher[1].InitAny(who:= aktData.counts^.RepeatedPublishsAfterPubrel,	Topic:= ADR(topics[1]), ValueName:= ADR(''), ValueDiff:= 0, DecimalPlace:= 0, QoS:= QoS.AtMostOnce, RetainMqtt:= TRUE, MinTime:= T#1S, MQTT_IN_OUT:= MQTT_IN_OUT);
	topics[2] := concat(STR1:= who.ClientID,STR2:='Supervision/RepeatedPubrel');
	publisher[2].InitAny(who:= aktData.counts^.RepeatedPubrel, Topic:= ADR(topics[2]), ValueName:= ADR(''), ValueDiff:= 0, DecimalPlace:= 0, QoS:= QoS.AtMostOnce, RetainMqtt:= TRUE, MinTime:= T#1S, MQTT_IN_OUT:= MQTT_IN_OUT);
	topics[3] := concat(STR1:= who.ClientID,STR2:='Supervision/CountRepeatedPing');
	publisher[3].InitAny(who:= aktData.counts^.CountRepeatedPing, Topic:= ADR(topics[3]), ValueName:= ADR(''), ValueDiff:= 0, DecimalPlace:= 0, QoS:= QoS.AtMostOnce, RetainMqtt:= TRUE, MinTime:= T#1S, MQTT_IN_OUT:= MQTT_IN_OUT);
	topics[4] := concat(STR1:= who.ClientID,STR2:='Supervision/CountRepeatedPingDisconnect');
	publisher[4].InitAny(who:= aktData.counts^.CountRepeatedPingDisconnect,	Topic:= ADR(topics[4]), ValueName:= ADR(''), ValueDiff:= 0, DecimalPlace:= 0, QoS:= QoS.AtMostOnce, RetainMqtt:= TRUE, MinTime:= T#1S, MQTT_IN_OUT:= MQTT_IN_OUT);
	topics[5] := concat(STR1:= who.ClientID,STR2:='Supervision/CountToBigTopics');
	publisher[5].InitAny(who:= aktData.counts^.CountToBigTopics, Topic:= ADR(topics[5]), ValueName:= ADR(''), ValueDiff:= 0, DecimalPlace:= 0, QoS:= QoS.AtMostOnce, RetainMqtt:= TRUE, MinTime:= T#1S, MQTT_IN_OUT:= MQTT_IN_OUT);
	topics[6] := concat(STR1:= who.ClientID,STR2:='Supervision/CountLengthErrors');
	publisher[6].InitAny(who:= aktData.counts^.CountLengthErrors, Topic:= ADR(topics[6]), ValueName:= ADR(''), ValueDiff:= 0, DecimalPlace:= 0, QoS:= QoS.AtMostOnce, RetainMqtt:= TRUE, MinTime:= T#1S, MQTT_IN_OUT:= MQTT_IN_OUT);
	topics[7] := concat(STR1:= who.ClientID,STR2:='Supervision/CountRepeatPublishReceive');
	publisher[7].InitAny(who:= aktData.counts^.CountRepeatPublishReceive, Topic:= ADR(topics[7]), ValueName:= ADR(''), ValueDiff:= 0, DecimalPlace:= 0, QoS:= QoS.AtMostOnce, RetainMqtt:= TRUE, MinTime:= T#1S, MQTT_IN_OUT:= MQTT_IN_OUT);
	topics[8] := concat(STR1:= who.ClientID,STR2:='Supervision/CountReceivedPublishs');
	publisher[8].InitAny(who:= aktData.counts^.CountReceivedPublishs, Topic:= ADR(topics[8]), ValueName:= ADR(''), ValueDiff:= 0, DecimalPlace:= 0, QoS:= QoS.AtMostOnce, RetainMqtt:= TRUE, MinTime:= T#1S, MQTT_IN_OUT:= MQTT_IN_OUT);
	topics[9] := concat(STR1:= who.ClientID,STR2:='Supervision/CountSendedPublishs');
	publisher[9].InitAny(who:= aktData.counts^.CountSendedPublishs,	Topic:= ADR(topics[9]), ValueName:= ADR(''), ValueDiff:= 0, DecimalPlace:= 0, QoS:= QoS.AtMostOnce, RetainMqtt:= TRUE, MinTime:= T#1S, MQTT_IN_OUT:= MQTT_IN_OUT);
	topics[10] := concat(STR1:= who.ClientID,STR2:='Supervision/CountRepeatSubscribe');
	publisher[10].InitAny(who:= aktData.counts^.CountRepeatSubscribe, Topic:= ADR(topics[10]), ValueName:= ADR(''), ValueDiff:= 0, DecimalPlace:= 0, QoS:= QoS.AtMostOnce, RetainMqtt:= TRUE, MinTime:= T#1S, MQTT_IN_OUT:= MQTT_IN_OUT);
	topics[11] := concat(STR1:= who.ClientID,STR2:='Supervision/CountRepeatUnsubscribe');
	publisher[11].InitAny(who:= aktData.counts^.CountRepeatUnsubscribe, Topic:= ADR(topics[11]), ValueName:= ADR(''), ValueDiff:= 0, DecimalPlace:= 0, QoS:= QoS.AtMostOnce, RetainMqtt:= TRUE, MinTime:= T#1S, MQTT_IN_OUT:= MQTT_IN_OUT);
	topics[12] := concat(STR1:= who.ClientID,STR2:='Supervision/CountRepeatetPubrec');
	publisher[12].InitAny(who:= aktData.counts^.CountRepeatetPubrec, Topic:= ADR(topics[12]), ValueName:= ADR(''), ValueDiff:= 0, DecimalPlace:= 0, QoS:= QoS.AtMostOnce, RetainMqtt:= TRUE, MinTime:= T#1S, MQTT_IN_OUT:= MQTT_IN_OUT);
	topics[13] := concat(STR1:= who.ClientID,STR2:='Supervision/RepeatedPublish');
	publisher[13].InitAny(who:= aktData.counts^.RepeatedPublish, Topic:= ADR(topics[13]), ValueName:= ADR(''), ValueDiff:= 0, DecimalPlace:= 0, QoS:= QoS.AtMostOnce, RetainMqtt:= TRUE, MinTime:= T#1S, MQTT_IN_OUT:= MQTT_IN_OUT);
	topics[14] := concat(STR1:= who.ClientID,STR2:='Supervision/CountOutputPublishCalled');
	publisher[14].InitAny(who:= aktData.counts^.CountOutputPublishCalled, Topic:= ADR(topics[14]), ValueName:= ADR(''), ValueDiff:= 0, DecimalPlace:= 0, QoS:= QoS.AtMostOnce, RetainMqtt:= TRUE, MinTime:= T#1S, MQTT_IN_OUT:= MQTT_IN_OUT);
	topics[15] := concat(STR1:= who.ClientID,STR2:='Supervision/CountReceivePubrelUnknown');
	publisher[15].InitAny(who:= aktData.counts^.CountReceivePubrelUnknown, Topic:= ADR(topics[15]), ValueName:= ADR(''), ValueDiff:= 0, DecimalPlace:= 0, QoS:= QoS.AtMostOnce, RetainMqtt:= TRUE, MinTime:= T#1S, MQTT_IN_OUT:= MQTT_IN_OUT);
	topics[16] := concat(STR1:= who.ClientID,STR2:='Supervision/CountReceiveUnsubackUnknown');
	publisher[16].InitAny(who:= aktData.counts^.CountReceiveUnsubackUnknown, Topic:= ADR(topics[16]), ValueName:= ADR(''), ValueDiff:= 0, DecimalPlace:= 0, QoS:= QoS.AtMostOnce, RetainMqtt:= TRUE, MinTime:= T#1S, MQTT_IN_OUT:= MQTT_IN_OUT);
	topics[17] := concat(STR1:= who.ClientID,STR2:='Supervision/CountReceiveSubackUnknown');
	publisher[17].InitAny(who:= aktData.counts^.CountReceiveSubackUnknown, Topic:= ADR(topics[17]), ValueName:= ADR(''), ValueDiff:= 0, DecimalPlace:= 0, QoS:= QoS.AtMostOnce, RetainMqtt:= TRUE, MinTime:= T#1S, MQTT_IN_OUT:= MQTT_IN_OUT);
	topics[18] := concat(STR1:= who.ClientID,STR2:='Supervision/CountReceivePubackUnknown');
	publisher[18].InitAny(who:= aktData.counts^.CountReceivePubackUnknown, Topic:= ADR(topics[18]), ValueName:= ADR(''), ValueDiff:= 0, DecimalPlace:= 0, QoS:= QoS.AtMostOnce, RetainMqtt:= TRUE, MinTime:= T#1S, MQTT_IN_OUT:= MQTT_IN_OUT);
	topics[19] := concat(STR1:= who.ClientID,STR2:='Supervision/CountReceivePubrecUnknown');
	publisher[19].InitAny(who:= aktData.counts^.CountReceivePubrecUnknown, Topic:= ADR(topics[19]), ValueName:= ADR(''), ValueDiff:= 0, DecimalPlace:= 0, QoS:= QoS.AtMostOnce, RetainMqtt:= TRUE, MinTime:= T#1S, MQTT_IN_OUT:= MQTT_IN_OUT);
	topics[20] := concat(STR1:= who.ClientID,STR2:='Supervision/CountReceivePubcompUnknown');
	publisher[20].InitAny(who:= aktData.counts^.CountReceivePubcompUnknown, Topic:= ADR(topics[20]), ValueName:= ADR(''), ValueDiff:= 0, DecimalPlace:= 0, QoS:= QoS.AtMostOnce, RetainMqtt:= TRUE, MinTime:= T#1S, MQTT_IN_OUT:= MQTT_IN_OUT);
	topics[21] := concat(STR1:= who.ClientID,STR2:='Supervision/CountReceivePubackUnknown');
	publisher[21].InitAny(who:= aktData.counts^.CountReceivePubackUnknown, Topic:= ADR(topics[21]), ValueName:= ADR(''), ValueDiff:= 0, DecimalPlace:= 0, QoS:= QoS.AtMostOnce, RetainMqtt:= TRUE, MinTime:= T#1S, MQTT_IN_OUT:= MQTT_IN_OUT);
	topics[22] := concat(STR1:= who.ClientID,STR2:='Supervision/CountBufferMoves');
	publisher[22].InitAny(who:= aktData.counts^.CountBufferMoves, Topic:= ADR(topics[22]), ValueName:= ADR(''), ValueDiff:= 0, DecimalPlace:= 0, QoS:= QoS.AtMostOnce, RetainMqtt:= TRUE, MinTime:= T#1S, MQTT_IN_OUT:= MQTT_IN_OUT);
	topics[23] := concat(STR1:= who.ClientID,STR2:='Supervision/CountNothingSend');
	publisher[23].InitAny(who:= aktData.counts^.CountNothingSend, Topic:= ADR(topics[23]), ValueName:= ADR(''), ValueDiff:= 0, DecimalPlace:= 0, QoS:= QoS.AtMostOnce, RetainMqtt:= TRUE, MinTime:= T#1S, MQTT_IN_OUT:= MQTT_IN_OUT);
	topics[24] := concat(STR1:= who.ClientID,STR2:='Supervision/CountConnectAttempt');
	publisher[24].InitAny(who:= aktData.counts^.CountConnectAttempt, Topic:= ADR(topics[24]), ValueName:= ADR(''), ValueDiff:= 0, DecimalPlace:= 0, QoS:= QoS.AtMostOnce, RetainMqtt:= TRUE, MinTime:= T#1S, MQTT_IN_OUT:= MQTT_IN_OUT);
	topics[25] := concat(STR1:= who.ClientID,STR2:='Supervision/CountSplitTopicSizeExceeded');
	publisher[25].InitAny(who:= aktData.counts^.CountSplitTopicSizeExceeded, Topic:= ADR(topics[25]), ValueName:= ADR(''), ValueDiff:= 0, DecimalPlace:= 0, QoS:= QoS.AtMostOnce, RetainMqtt:= TRUE, MinTime:= T#1S, MQTT_IN_OUT:= MQTT_IN_OUT);
	topics[26] := concat(STR1:= who.ClientID,STR2:='Supervision/CountWaitForRestOfPaket');
	publisher[26].InitAny(who:= aktData.counts^.CountWaitForRestOfPaket, Topic:= ADR(topics[26]), ValueName:= ADR(''), ValueDiff:= 0, DecimalPlace:= 0, QoS:= QoS.AtMostOnce, RetainMqtt:= TRUE, MinTime:= T#1S, MQTT_IN_OUT:= MQTT_IN_OUT);
	topics[27] := concat(STR1:= who.ClientID,STR2:='Supervision/CountResetBufferIn');
	publisher[27].InitAny(who:= aktData.counts^.CountResetBufferIn, Topic:= ADR(topics[27]), ValueName:= ADR(''), ValueDiff:= 0, DecimalPlace:= 0, QoS:= QoS.AtMostOnce, RetainMqtt:= TRUE, MinTime:= T#1S, MQTT_IN_OUT:= MQTT_IN_OUT);
	topics[28] := concat(STR1:= who.ClientID,STR2:='Supervision/InBufferMoved');
	publisher[28].InitAny(who:= aktData.counts^.InBufferMoved, Topic:= ADR(topics[28]), ValueName:= ADR(''), ValueDiff:= 0, DecimalPlace:= 0, QoS:= QoS.AtMostOnce, RetainMqtt:= TRUE, MinTime:= T#1S, MQTT_IN_OUT:= MQTT_IN_OUT);
	topics[29] := concat(STR1:= who.ClientID,STR2:='Supervision/CountOutSendNotFree');
	publisher[29].InitAny(who:= aktData.counts^.CountOutSendNotFree, Topic:= ADR(topics[29]), ValueName:= ADR(''), ValueDiff:= 0, DecimalPlace:= 0, QoS:= QoS.AtMostOnce, RetainMqtt:= TRUE, MinTime:= T#1S, MQTT_IN_OUT:= MQTT_IN_OUT);
	topics[30] := concat(STR1:= who.ClientID,STR2:='Supervision/CountInSendNotFree');
	publisher[30].InitAny(who:= aktData.counts^.CountInSendNotFree, Topic:= ADR(topics[30]), ValueName:= ADR(''), ValueDiff:= 0, DecimalPlace:= 0, QoS:= QoS.AtMostOnce, RetainMqtt:= TRUE, MinTime:= T#1S, MQTT_IN_OUT:= MQTT_IN_OUT);
	topics[31] := concat(STR1:= who.ClientID,STR2:='Supervision/CountCantSendPublishBufferToFull');
	publisher[31].InitAny(who:= aktData.counts^.CountCantSendPublishBufferToFull, Topic:= ADR(topics[31]), ValueName:= ADR(''), ValueDiff:= 0, DecimalPlace:= 0, QoS:= QoS.AtMostOnce, RetainMqtt:= TRUE, MinTime:= T#1S, MQTT_IN_OUT:= MQTT_IN_OUT);
	topics[32] := concat(STR1:= who.ClientID,STR2:='Supervision/CountUnkownPaket');
	publisher[32].InitAny(who:= aktData.counts^.CountUnkownPaket, Topic:= ADR(topics[32]), ValueName:= ADR(''), ValueDiff:= 0, DecimalPlace:= 0, QoS:= QoS.AtMostOnce, RetainMqtt:= TRUE, MinTime:= T#1S, MQTT_IN_OUT:= MQTT_IN_OUT);
	topics[33] := concat(STR1:= who.ClientID,STR2:='Supervision/SendedBytes');
	publisher[33].InitAny(who:= aktData.counts^.SendedBytes, Topic:= ADR(topics[33]), ValueName:= ADR(''), ValueDiff:= 0, DecimalPlace:= 0, QoS:= QoS.AtMostOnce, RetainMqtt:= TRUE, MinTime:= T#1S, MQTT_IN_OUT:= MQTT_IN_OUT);
	topics[34] := concat(STR1:= who.ClientID,STR2:='Supervision/ReceivedBytes');
	publisher[34].InitAny(who:= aktData.counts^.ReceivedBytes, Topic:= ADR(topics[34]), ValueName:= ADR(''), ValueDiff:= 0, DecimalPlace:= 0, QoS:= QoS.AtMostOnce, RetainMqtt:= TRUE, MinTime:= T#1S, MQTT_IN_OUT:= MQTT_IN_OUT);
	topics[35] := concat(STR1:= who.ClientID,STR2:='Supervision/InSlotsWorking');
	publisher[35].InitAny(who:= aktData.counts^.InSlotsWorking, Topic:= ADR(topics[35]), ValueName:= ADR(''), ValueDiff:= 0, DecimalPlace:= 0, QoS:= QoS.AtMostOnce, RetainMqtt:= TRUE, MinTime:= T#1S, MQTT_IN_OUT:= MQTT_IN_OUT);
	topics[36] := concat(STR1:= who.ClientID,STR2:='Supervision/OutSlotsWorking');
	publisher[36].InitAny(who:= aktData.counts^.OutSlotsWorking, Topic:= ADR(topics[36]), ValueName:= ADR(''), ValueDiff:= 0, DecimalPlace:= 0, QoS:= QoS.AtMostOnce, RetainMqtt:= TRUE, MinTime:= T#1S, MQTT_IN_OUT:= MQTT_IN_OUT);
	topics[37] := concat(STR1:= who.ClientID,STR2:='Supervision/DynMemUsagePointer');
	publisher[37].InitAny(who:= aktData.counts^.DynMemUsagePointer, Topic:= ADR(topics[37]), ValueName:= ADR(''), ValueDiff:= 0, DecimalPlace:= 0, QoS:= QoS.AtMostOnce, RetainMqtt:= TRUE, MinTime:= T#1S, MQTT_IN_OUT:= MQTT_IN_OUT);
	topics[38] := concat(STR1:= who.ClientID,STR2:='Supervision/MqttsDoneIo');
	publisher[38].InitAny(who:= aktData.counts^.MqttsDoneIo, Topic:= ADR(topics[38]), ValueName:= ADR(''), ValueDiff:= 0, DecimalPlace:= 0, QoS:= QoS.AtMostOnce, RetainMqtt:= TRUE, MinTime:= T#1S, MQTT_IN_OUT:= MQTT_IN_OUT);
	topics[39] := concat(STR1:= who.ClientID,STR2:='Supervision/PerSecond/PublishsSend');
	publisher[39].InitAny(who:= aktData.counts^.PublishsSendPerSeconde, Topic:= ADR(topics[39]), ValueName:= ADR(''), ValueDiff:= 0, DecimalPlace:= 0, QoS:= QoS.AtMostOnce, RetainMqtt:= TRUE, MinTime:= T#1S, MQTT_IN_OUT:= MQTT_IN_OUT);
	publisher[39].SetTrigger(which:= aktData.secImp);
	topics[40] := concat(STR1:= who.ClientID,STR2:='Supervision/PerSecond/PublishsReceived');
	publisher[40].InitAny(who:= aktData.counts^.PublishsReceivedPerSeconde, Topic:= ADR(topics[40]), ValueName:= ADR(''), ValueDiff:= 0, DecimalPlace:= 0, QoS:= QoS.AtMostOnce, RetainMqtt:= TRUE, MinTime:= T#1S, MQTT_IN_OUT:= MQTT_IN_OUT);
	publisher[40].SetTrigger(which:= aktData.secImp);
	topics[41] := concat(STR1:= who.ClientID,STR2:='Supervision/PerSecond/SendedBytes');
	publisher[41].InitAny(who:= SendedBytesPerSecond, Topic:= ADR(topics[41]), ValueName:= ADR(''), ValueDiff:= 0, DecimalPlace:= 0, QoS:= QoS.AtMostOnce, RetainMqtt:= TRUE, MinTime:= T#1S, MQTT_IN_OUT:= MQTT_IN_OUT);
	publisher[41].SetTrigger(which:= aktData.secImp);
	topics[42] := concat(STR1:= who.ClientID,STR2:='Supervision/PerSecond/ReceivedBytes');
	publisher[42].InitAny(who:= ReceivedBytesPerSecond, Topic:= ADR(topics[42]), ValueName:= ADR(''), ValueDiff:= 0, DecimalPlace:= 0, QoS:= QoS.AtMostOnce, RetainMqtt:= TRUE, MinTime:= T#1S, MQTT_IN_OUT:= MQTT_IN_OUT);
	publisher[42].SetTrigger(which:= aktData.secImp);
	topics[43] := concat(STR1:= who.ClientID,STR2:=concat(STR1:='Supervision/Per', STR2:=  concat(STR1:= perXTopic, STR2:='/SendedBytes')));
	publisher[43].InitAny(who:= SendedBytesPerX, Topic:= ADR(topics[43]), ValueName:= ADR(''), ValueDiff:= 0, DecimalPlace:= 0, QoS:= QoS.AtMostOnce, RetainMqtt:= TRUE, MinTime:= T#1S, MQTT_IN_OUT:= MQTT_IN_OUT);
	publisher[43].SetTrigger(which:= ADR(TriggerX));
	topics[44] := concat(STR1:= who.ClientID,STR2:=concat(STR1:='Supervision/Per', STR2:=  concat(STR1:= perXTopic, STR2:='/ReceivedBytes')));
	publisher[44].InitAny(who:= ReceivedBytesPerX, Topic:= ADR(topics[44]), ValueName:= ADR(''), ValueDiff:= 0, DecimalPlace:= 0, QoS:= QoS.AtMostOnce, RetainMqtt:= TRUE, MinTime:= T#1S, MQTT_IN_OUT:= MQTT_IN_OUT);
	publisher[44].SetTrigger(which:= ADR(TriggerX));
	topics[45] := concat(STR1:= who.ClientID,STR2:=concat(STR1:='Supervision/Per', STR2:=  concat(STR1:= perXTopic, STR2:='/PublishsSend')));
	publisher[45].InitAny(who:= PublishSendPerX, Topic:= ADR(topics[45]), ValueName:= ADR(''), ValueDiff:= 0, DecimalPlace:= 0, QoS:= QoS.AtMostOnce, RetainMqtt:= TRUE, MinTime:= T#1S, MQTT_IN_OUT:= MQTT_IN_OUT);
	publisher[45].SetTrigger(which:= ADR(TriggerX));
	topics[46] := concat(STR1:= who.ClientID,STR2:=concat(STR1:='Supervision/Per', STR2:=  concat(STR1:= perXTopic, STR2:='/PublishsReceived')));
	publisher[46].InitAny(who:= PublishReceivedPerX, Topic:= ADR(topics[46]), ValueName:= ADR(''), ValueDiff:= 0, DecimalPlace:= 0, QoS:= QoS.AtMostOnce, RetainMqtt:= TRUE, MinTime:= T#1S, MQTT_IN_OUT:= MQTT_IN_OUT);
	publisher[46].SetTrigger(which:= ADR(TriggerX));
	
	FOR i := 0 TO COUNT_PUBLISHER - 1 DO
		publisher[i].PayloadStartup := TRUE;
	END_FOR
	
END_IF
MQTT_IN_OUT.clientFB(
	MQTT_IN_OUT:= MQTT_IN_OUT, 
	ENABLE:= TRUE, 
	URL:= lBroker, 
	TIMEOUT:= T#5S);

//Send Data at X time
tc := DWORD_TO_TIME(tx - tl);
TriggerX := FALSE;
IF NOT who.BROKER_CONNECTED THEN
	SendedBytesPerSecondLast := 0;
	ReceivedBytesPerSecondLast := 0;
	SendedBytesPerXLast := 0;
	ReceivedBytesPerXLast := 0;

END_IF
IF tc > TimeX THEN
	tl := tx;
	TriggerX := TRUE;
	SendedBytesPerX := TO_UDINT(aktData.counts^.SendedBytes - SendedBytesPerXLast);
	SendedBytesPerXLast := aktData.counts^.SendedBytes;
	ReceivedBytesPerX := TO_UDINT(aktData.counts^.ReceivedBytes - ReceivedBytesPerXLast);
	ReceivedBytesPerXLast := aktData.counts^.ReceivedBytes;
	PublishSendPerX := TO_UINT(aktData.counts^.CountSendedPublishs - PublishSendPerXLast);
	PublishSendPerXLast := aktData.counts^.CountSendedPublishs;
	PublishReceivedPerX := TO_UINT(aktData.counts^.CountReceivedPublishs - PublishReceivedPerXLast);
	PublishReceivedPerXLast := aktData.counts^.CountReceivedPublishs;
END_IF;

IF aktdata.secImp^ THEN
	SendedBytesPerSecond := TO_UDINT(aktData.counts^.SendedBytes - SendedBytesPerSecondLast);
	SendedBytesPerSecondLast := aktData.counts^.SendedBytes;
	ReceivedBytesPerSecond := TO_UDINT(aktData.counts^.ReceivedBytes - ReceivedBytesPerSecondLast);
	ReceivedBytesPerSecondLast := aktData.counts^.ReceivedBytes;	
END_IF
FOR i := 0 TO 46 DO
	publisher[i]();
END_FOR
IF aktData.ErrorHistory <> 0 AND_THEN (OldHistoryNum <> aktData.ErrorHistory^[0].nr) AND NOT SendHistroy THEN
	//now publish all new errors...
	//first search oldest not send error
	LastHistoryFound := FALSE;
	FOR i := 0 TO aktData.CountHistoryItems - 1 DO
		IF aktData.ErrorHistory^[i].nr = OldHistoryNum THEN
			i := i - 1;
			LastHistoryFound := TRUE;
			EXIT;
		END_IF
	END_FOR
	IF NOT LastHistoryFound THEN
		//last elemenet was not found. start with previus
		i := aktData.CountHistoryItems - 2;
	END_IF	
	OldHistoryNum := aktData.ErrorHistory^[i].nr;
	HistoryJSON.error.AsString := TO_STRING(aktData.ErrorHistory^[i].error);
	HistoryJSON.DoesDisconnect.Boolean := aktData.ErrorHistory^[i].DoesDisconnect;
	HistoryJSON.when.AsDateTime := aktData.ErrorHistory^[i].when;
	HistoryJSON.nr.Integer := aktData.ErrorHistory^[i].nr;
	HistoryJSON.ERROR_C.Integer := TO_DINT(aktData.ErrorHistory^[i].ERROR_C);
	HistoryJSON.ERROR_T.Integer := aktData.ErrorHistory^[i].ERROR_T;
	HistoryJSON.text.AsString := aktData.ErrorHistory^[i].text;
	HistoryJSON.MqttsDoneIo.Integer := TO_DINT(aktData.ErrorHistory^[i].MqttsDoneIo);
	HistoryJSON.SendedBytes.Integer := TO_DINT(aktData.ErrorHistory^[i].SendedBytes);
	HistoryJSON.ReceivedBytes.Integer := TO_DINT(aktData.ErrorHistory^[i].ReceivedBytes);
	HistoryJSON.ResultSend.Integer := TO_DINT(aktData.ErrorHistory^[i].ResultSend);
	HistoryJSON.ResultReceive.Integer := TO_DINT(aktData.ErrorHistory^[i].ResultReceive);
	toJSON.Execute := TRUE;
		
END_IF
toJSON(JSONString:= ADR(HistoryString), 
	JSONStringSize:= SIZEOF(HistoryString), 
	JSONVars:= ADR(HistoryJSON), 
	NumberOfVars:= SIZEOF(HistoryJSON)/SIZEOF(JSONVAR),
	MaxLevel:= 1);
IF toJSON.done THEN
	toJSON.Execute := FALSE;
	toJSON();
	SendHistroy := TRUE;
END_IF
HistoryPublisher(
	Topic:= ADR(HistoryTopic), 
	PayloadString:= ADR(HistoryString), 
	PublishAsString:= TRUE,
	QoSIn:= QoS.AtLeastOnce, 
	send:= SendHistroy,
	MRetain:= TRUE);
IF HistoryPublisher.done THEN
	SendHistroy := FALSE;
	HistoryPublisher(send:= SendHistroy);
END_IF

END_FUNCTION_BLOCK

// MQTT/TestCases/TestBigPacket
FUNCTION_BLOCK TestBigPacket
VAR_INPUT
	url:STRING:='test.mosquitto.org';
END_VAR
VAR_OUTPUT
	MQTT_IN_OUT:POINTER TO MQTT_IN_OUT;
END_VAR
VAR
	in_out:MQTT_IN_OUT;
	SendBuffer:ARRAY[0..SIZE_OF_PAKET]OF BYTE;
	//ReceiveBuffer:ARRAY[0..SIZE_OF_PAKET]OF BYTE;
	init: BOOL;
	step:UINT;
	ts:USINT;
	i:UDINT;
	Pos:UDINT;
	breaker:UDINT;

	send: BOOL;
	publisher:MqttPublish;
	//handle:MqttClient;
	subscribe: BOOL;
	subscriber:MQTTSubscribe;
	checker:PayloadChecker;
	countReceivedOK:UINT;
	countReceivedNOK:UINT;
	rand:CommonTypesAndFunctions.Rand;
END_VAR
VAR CONSTANT
	SIZE_OF_PAKET:UDINT:=15000000;
	//SIZE_OF_PAKET:UDINT:=150000000;
	TOPIC:STRING:='SD_MQTT/TESTBIGPACKET';
END_VAR

IF NOT init THEN
	init := TRUE;
	in_out.COM_CONFIG.MaxPayloadSize := SIZE_OF_PAKET;
	subscriber.SetMqttInOut(MQTT_IN_OUT:= in_out);
	publisher.SetMqttInOut(MQTT_IN_OUT:= in_out);
	in_out.ClientID := 'TestBIG';
END_IF

CASE step OF
	0://Startup
		pos := 0;
		step := 2;
		//do some stuff on the payload
		ts := TO_BYTE(rand.getRand(LowIn:=0, HighIn:= 255));
		
		
	2://do data
		FOR breaker := 0 TO 100000 DO
			SendBuffer[Pos] := ts;
			ts := ts + 1;
			IF Pos >= SIZE_OF_PAKET - 1 THEN
				step := 10;
				EXIT;
			END_IF	
			Pos := Pos + 1;
		END_FOR 
	10://publish this packet
		send := TRUE;
		step := 20;
	20://wait to send be done
		IF publisher.done THEN
			send := FALSE;
			step := 30;
		END_IF
	30://now get the data back...
		subscribe := TRUE;
		step := 40;
	40://wait subscription is done
		IF subscriber.SubscribeDone THEN
			step:=50;
		END_IF
	50://wait payload is received
		IF checker.received THEN
			IF checker.testIO THEN
				countReceivedOK := countReceivedOK + 1;
			ELSE
				countReceivedNOK := countReceivedNOK + 1;
			END_IF
			subscribe := FALSE;
			//next run:
			step:=0;
		END_IF
END_CASE
checker(with:=ADR(SendBuffer), size:= SIZE_OF_PAKET);
subscriber(
	Topic:= ADR(TOPIC), 
	QoSSubscribe:= QoS.ExactlyOnce, 
	ExpectingString:= FALSE, 
	Callback:= checker);
	subscriber.subscribe:= subscribe;
publisher(
	Topic:= ADR(TOPIC), 
	Payload:= ADR(SendBuffer), 
	PayloadLength:= SIZE_OF_PAKET, 
	QoSIn:=QoS.ExactlyOnce , 
	MRetain:= TRUE, 
	send:= send);
	
in_out.clientFB(
	MQTT_IN_OUT:= in_out, 
	ENABLE:= TRUE, 
	URL:= url, 
	TIMEOUT:= T#5S);

//FB_Init ist immer implizit verfügbar und wird primär für die Initialisierung verwendet.
//Der Rückgabewert wird nicht ausgewertet. Für gezielte Einflussnahme können Sie
//die Methoden explizit deklarieren und darin mit dem Standard-Initialisierungscode 
//zusätzlichen Code bereitstellen. Sie können den Rückgabewert auswerten.
METHOD FB_Init: BOOL
VAR_INPUT    
bInitRetains: BOOL; // TRUE: Die Retain-Variablen werden initialisiert (Reset warm / Reset kalt)    
bInCopyCode: BOOL;  // TRUE: Die Instanz wird danach in den Kopiercode kopiert (Online-Change)
END_VAR
MQTT_IN_OUT := adr(in_out);
END_METHOD

END_FUNCTION_BLOCK

// MQTT/TestCases/Test Interfaces/PayloadChecker
FUNCTION_BLOCK PayloadChecker IMPLEMENTS MQTT_SUBSCRIBE_CALLBACK
VAR_INPUT
	with:POINTER TO BYTE;
	size:UDINT;
END_VAR
VAR_OUTPUT
	testIO: BOOL;
	received: BOOL;

END_VAR
VAR
	lwith:POINTER TO BYTE;
	lsize:UDINT;
END_VAR

lwith := with;
lsize := size;
testIO := FALSE;
received := FALSE;

METHOD PublishReceived : BOOL
VAR_INPUT
	(*Collection of received Data*)
	Data	: CALLBACK_DATA;
END_VAR
VAR 
	i:UDINT;
END_VAR
received := TRUE;
IF lsize <> Data.PayloadSize THEN
	testio := FALSE;
	RETURN;
END_IF
FOR i := 0 TO lsize DO
	IF lwith[i] <> Data.Payload[i] THEN
		RETURN;
	END_IF
END_FOR

testio := TRUE;
END_METHOD

END_FUNCTION_BLOCK

// MQTT/TestCases/TestNestedSubscriber
FUNCTION_BLOCK TestNestedSubscriber
VAR_INPUT
END_VAR
VAR_OUTPUT
END_VAR
VAR
	MQTT_IN_OUT:MQTT_IN_OUT;
	init: BOOL;
	subscriber:REFERENCE TO MQTTSubscribeNested;
	callback:CallbackCollector;
	StringReceiver:SingelStringCallback;
	ReceiveTopic:STRING(255);
	ReceivePayload:STRING(255);
	subscribe: BOOL := TRUE;

END_VAR

IF NOT init THEN
	init:= TRUE;

END_IF
MQTT_IN_OUT.clientFB(URL:= 'test.mosquitto.org', ENABLE:= TRUE, TIMEOUT:= T#5S, MQTT_IN_OUT:= MQTT_IN_OUT);
subscriber.subscribe := subscribe;

//FB_Init ist immer implizit verfügbar und wird primär für die Initialisierung verwendet.
//Der Rückgabewert wird nicht ausgewertet. Für gezielte Einflussnahme können Sie
//die Methoden explizit deklarieren und darin mit dem Standard-Initialisierungscode 
//zusätzlichen Code bereitstellen. Sie können den Rückgabewert auswerten.
METHOD FB_Init: BOOL
VAR_INPUT    
bInitRetains: BOOL; // TRUE: Die Retain-Variablen werden initialisiert (Reset warm / Reset kalt)    
bInCopyCode: BOOL;  // TRUE: Die Instanz wird danach in den Kopiercode kopiert (Online-Change)
END_VAR


	subscriber REF= MQTT_IN_OUT.clientFB.GetSubscriber();
	subscriber.Callback := callback;
	subscriber.ExpectingString := TRUE;
	subscriber.subscribe := TRUE;
	subscriber.Topic := ADR('test/#');
	StringReceiver.Init(payload:= ADR(ReceivePayload), topic:= ADR(ReceiveTopic));
	callback.put(instance:= StringReceiver);
END_METHOD

END_FUNCTION_BLOCK
